ELSE
	(* server device not ready, reset local ready flag *)
	bReady := FALSE;
	nErrorId := BACnet_ERR_OPERATIONAL;
END_IF
(* set error flag *)
bError := (nErrorId <> BACnet_ERR_NO_ERROR);
END_FUNCTION_BLOCK

(* POU FB_BACnet_PulseConverter_RAW, ST *)
FUNCTION_BLOCK FB_BACnet_PulseConverter_RAW
VAR_INPUT
	nRawIn			AT%Q*: UINT; (* ~(BACnet_RawIoPulseConverterUnsignedValue : : ) *)
	bNoSensor		: BOOL;
	bOverRange		: BOOL;
	bUnderRange		: BOOL;
	bOpenLoop		: BOOL;
	bShortedLoop	: BOOL;
	bCommFailure	: BOOL;
	bConfigError	: BOOL;
	bOtherFault		: BOOL;
END_VAR
VAR_IN_OUT
	Device			: FB_BACnet_Device;
END_VAR
VAR_OUTPUT
	bReady			: BOOL;
	fPresentValue	: REAL;
	nCount			: UDINT;
	bOverridden		: BOOL;
	bOutOfService	: BOOL;
	bFault			: BOOL;
	bInAlarm		: BOOL;
	bError			: BOOL;
	nErrorId		: UINT;
END_VAR
VAR
	_PresentValueIn AT%I*: REAL; 	(* ~(BACnet_PresentValue 		:		: )
								   		(BACnet_ObjectType 			: PC	: )
										(BACnet_InputReference		: 		: nolink, disable) *)
	_Count AT%I*: UDINT;			(* ~(BACnet_Count		 		:		: ) *)
	_ObjectId AT%I*: DWORD;			(* ~(BACnet_ObjectIdentifier	:		: LINK) *)
	_StatusFlags AT%I*: WORD; 		(* ~(BACnet_StatusFlags 		:		: )	*)
	_ReliabilityIn AT%I*: WORD;		(* ~(BACnet_Reliability 		:		: )	*)
	_ReliabilityOut AT%Q*: WORD := BACnetReliability_no_fault_detected;(* ~(BACnet_Reliability 	:		: )	*)
	_StatusFlagsBits : ST_BACnet_StatusFlags;
	_nUpdateCount : UDINT := 0;
END_VAR
(* update server device *)
IF (Device._nUpdateCount = _nUpdateCount) THEN
	Device();
END_IF
(* remind current number of update counter *)
_nUpdateCount := Device._nUpdateCount;

(* handle raw error *)
IF (_ReliabilityIn <> BACnetReliability_configuration_error) THEN
	IF bNoSensor THEN
		_ReliabilityOut := BACnetReliability_no_sensor;
	ELSIF bOverRange THEN
		_ReliabilityOut := BACnetReliability_over_range;
	ELSIF bUnderRange THEN
		_ReliabilityOut := BACnetReliability_under_range;
	ELSIF bOpenLoop THEN
		_ReliabilityOut := BACnetReliability_open_loop;
	ELSIF bShortedLoop THEN
		_ReliabilityOut := BACnetReliability_shorted_loop;
	ELSIF bCommFailure THEN
		_ReliabilityOut := BACnetReliability_communication_failure;
	ELSIF bOtherFault THEN
		_ReliabilityOut := BACnetReliability_unreliable_other;
	ELSE
		_ReliabilityOut := BACnetReliability_no_fault_detected;
	END_IF
ELSE
	_ReliabilityOut := BACnetReliability_no_fault_detected;
END_IF

IF Device.bFirstCycle THEN
	(* first call of the server device since reboot/reset *)
	bReady := FALSE;

ELSIF (_StatusFlags < 4) THEN
	(* wrong mapping *)
	nErrorId := BACnet_ERR_WRONG_MAPPING;
	bReady := FALSE;

ELSIF Device.bOperational THEN
	(* ready state *)
	bReady := TRUE;
	nErrorId := BACnet_ERR_NO_ERROR;

	(* present value *)
	fPresentValue := _PresentValueIn;

	(* build bit states *)
	_StatusFlagsBits := F_BACnet_StatusFlags(_StatusFlags);

	(* copy states to output *)
	bOverridden		:= _StatusFlagsBits.overridden;
	bOutOfService	:= _StatusFlagsBits.out_of_service;
	bFault			:= _StatusFlagsBits.fault;
	bInAlarm		:= _StatusFlagsBits.in_alarm;

	(* additional information *)
	nCount			:= _Count;

ELSE
	(* server device not ready, reset local ready flag *)
	bReady := FALSE;
	nErrorId := BACnet_ERR_OPERATIONAL;
END_IF
(* set error flag *)
bError := (nErrorId <> BACnet_ERR_NO_ERROR);
END_FUNCTION_BLOCK

(* POU FB_BACnet_PWM, ST *)
FUNCTION_BLOCK FB_BACnet_PWM
VAR_INPUT
	bEnable			: BOOL;
	fPercent		: REAL; (* 0...100% *)
	tPeriod			: TIME; (* PWM period time *)
END_VAR
VAR_OUTPUT
	bEnablePV		: BOOL;
	bPresentValue	: BOOL;
END_VAR
VAR
	_fOut			: REAL;
	_tOn			: TIME;
	_tonPeriod		: TON;
	_tofOn			: TOF;
END_VAR
(* check limits *)
_fOut := LIMIT(0.0, fPercent, 100.0);

(* convert from percent value to time value in relation to period time (100% = tPara_Period, 0% = 0s) *)
_tOn := REAL_TO_TIME((_fOut / 100.0) * TIME_TO_REAL(tPeriod));

(* call period timer *)
_tonPeriod(
	IN	:= TRUE,
	PT	:= tPeriod,
	Q	=> ,
	ET	=> );

(* call on timer *)
_tofOn(
	IN	:= _tonPeriod.Q AND (_tOn > T#0ms),
	PT	:= _tOn,
	Q	=> ,
	ET	=> );

IF _tonPeriod.Q THEN
	_tonPeriod(IN:= FALSE);
	_tonPeriod(IN:= TRUE);
END_IF

(* set output *)
bPresentValue := (_tofOn.Q OR _tofOn.IN) AND bEnable;
bEnablePV := bEnable;
END_FUNCTION_BLOCK

(* POU FB_BACnet_RecipientListProperty, ST *)
FUNCTION_BLOCK FB_BACnet_RecipientListProperty
VAR_INPUT
	tObjectID			: T_BACnet_ObjectIdentifier := 16#FFFFFFFF;
	bAutoGet			: BOOL:=TRUE; (* TRUE = get data from property when ADS connection OR object ID changed *)
	bGet				: BOOL; (* FALSE --> TRUE = get data from property *)
	bSet				: BOOL; (* FALSE --> TRUE = set data into property *)
END_VAR
VAR_IN_OUT
	stAdsConn			: ST_BACnet_AdsConnection;
	stRecipients		: ST_BACnet_RecipientListDevice;
END_VAR
VAR_OUTPUT
	bDone				: BOOL;
	bBusy				: BOOL;
	bError				: BOOL;
	nErrorId			: UINT;
END_VAR
VAR
	_fbReadProp		: FB_BACnet_ReadProp;
	_fbWriteProp	: FB_BACnet_WriteProp;
	_i				: INT;
	_rtrigGet		: R_TRIG;
	_rtrigSet		: R_TRIG;

	_nAdsReloadOld	: USINT;
	_tObjectIDOld	: T_BACnet_ObjectIdentifier := 16#FFFFFFFF;

	_iEntryCheck	: UDINT;
	_iEntry			: INT;
	_iDataEntry		: INT;
	_iReadElems		: UDINT;

	_pEntryList		: POINTER TO T_BACnet_DestinationDeviceArray;

	_cbDestList		: UDINT;
	_cbDestListElem	: UDINT;
END_VAR
(*
	enum BACnetRecipient_Choice
	{
	      device,
	      address
	};
	
	typedef struct _BACnetObjectIdentifier
	{
	      union
	      {
	            struct 
	            {
	                  DWORD objInst : 22;
	                  DWORD objType : 10;
	            };
	            DWORD objId;
	      };
	}BACnetObjectIdentifier, *PBACnetObjectIdentifier;
	
	typedef struct _BACnetAddress
	{
	      BACnetAddressChoice choice;
	      BYTE layerAddress[7]; // MS/TP...LonTalk 
	      BYTE reserved;
	      USHORT      network_number;
	}BACnetAddress, *PBACnetAddress;
	
	enum BACnetAddressChoice
	{
	      Ethernet,
	      Arcnet,
	      MsTp,
	      LonTalk,
	      LonTalkNeuronId,
	      Address_3,
	      Address_4,
	      Address_5,
	      Broadcast
	};
	
	typedef struct _BACnetRecipient
	{ 
	      BACnetRecipient_Choice choiceField;
	      union
	      {
	            BACnetObjectIdentifier  device;
	            BACnetAddress           address;
	      };
	}BACnetRecipient,*PBACnetRecipient;
		
	typedef struct _BACnetDestination
	{ 
	      ULONG                              validDays;  //Bitfield of BACnetDaysOfWeek
	      BACnetTime                         fromTime;
	      BACnetTime                         toTime;
	      BACnetRecipient                    recipient;
	      ULONG                              processIdentifier;
	      DWORD                              transitionsBits;  // BACnetEventTransitionBits
	      BOOL                               issueConfirmedNotifications;
	}BACnetDestination,*PBACnetDestination;


*)

(* ADS read *)
_fbReadProp(
	BACnetDevicePort	:= stAdsConn.nAmsPort,
	bExecute			:= ,
	sNetId				:= stAdsConn.sAmsNetId,
	ObjectType			:= F_BACnet_GetObjType(tObjectID),
	PropertyID			:= BACnetPropertyIdentifier_RecipientList,
	DataType			:= BACnetDataType_RecipientArr,
	ObjectInstance		:= F_BACnet_GetObjInstance(tObjectID),
	ptrValue			:= ADR(stBACnet_AdsBuffer.arrData),
	nLenValue			:= SIZEOF(stBACnet_AdsBuffer.arrData),
	bDone				=> ,
	bBusy				=> ,
	bError				=> ,
	nErrID				=> ,
	nProcessedLen		=> );

(* ADS write *)
_fbWriteProp(
	BACnetDevicePort	:= stAdsConn.nAmsPort,
	bExecute			:= ,
	sNetId				:= stAdsConn.sAmsNetId,
	ObjectType			:= F_BACnet_GetObjType(tObjectID),
	PropertyID			:= BACnetPropertyIdentifier_RecipientList,
	Priority			:= BACnetPriority_None,
	DataType			:= BACnetDataType_RecipientArr,
	ObjectInstance		:= F_BACnet_GetObjInstance(tObjectID),
	ptrValue			:= ADR(stBACnet_AdsBuffer.arrData),
	nLenValue			:= _iDataEntry * _cbDestListElem,
	bDone				=> ,
	bBusy				=> ,
	bError				=> ,
	nErrID				=> );

(* trigger start event *)
_rtrigGet(CLK:= bGet, Q=> );
_rtrigSet(CLK:= bSet, Q=> );

(* state machine *)
CASE _i OF

	0: (* Idle *)
		IF 		_rtrigGet.Q
			OR	_rtrigSet.Q
			OR	(		(		(_nAdsReloadOld <> stAdsConn.nReload)
							OR	(_tObjectIDOld <> tObjectID)
						)
					AND	bAutoGet
				)
		THEN
			IF (NOT stAdsConn.bValid) THEN
				(* ADS connection not valid *)
				nErrorId := BACnet_ERR_INVALID_ADS_CONN;
			ELSE
				(* decide get or set *)
				IF _rtrigGet.Q THEN
					_i := 1;
				ELSIF _rtrigSet.Q THEN
					_i := 11;
				ELSIF bAutoGet THEN
					_i := 1;
				END_IF
				nErrorId := BACnet_ERR_NO_ERROR;
				(* reset index *)
				_iEntry	:= 0;
				(* initialize pointer *)
				_pEntryList := ADR(stBACnet_AdsBuffer.arrData);
				(* remind parameter *)
				_tObjectIDOld := tObjectID;
				_nAdsReloadOld := stAdsConn.nReload;
			END_IF
			(* reset done flag *)
			bDone := FALSE;
		END_IF
		IF (NOT bGet) AND (NOT bSet) AND (NOT bAutoGet) THEN
			nErrorId := BACnet_ERR_NO_ERROR;
			bDone := FALSE;
		END_IF

	(* READ *)
	1: (* read object property data via ADS *)
		IF TestAndSet(stBACnet_AdsBuffer.bTestSet) THEN
			IF _fbReadProp.bExecute THEN
				IF _fbReadProp.bError THEN
					_i := 100;
					nErrorId := BACnet_ERR_ADS_Read;
					_fbReadProp.bExecute := FALSE;
				ELSIF (NOT _fbReadProp.bBusy) THEN
					_i := 2;
					_fbReadProp.bExecute := FALSE;
					(* clear output data *)
					MEMSET(ADR(stRecipients), 0, SIZEOF(stRecipients));
					(* check array size *)
					_cbDestList 	:= SIZEOF(_pEntryList^);
					_cbDestListElem	:= SIZEOF(_pEntryList^[0]);
					_iEntryCheck := MIN(_fbReadProp.nProcessedLen, _cbDestList) MOD _cbDestListElem;
					IF (_iEntryCheck <> 0) OR (_cbDestListElem = 0) THEN
						_i := 100;
						nErrorId := BACnet_ERR_ADS_WrongEntrySize;
					ELSE
						(* scan property *)
						_iDataEntry := 0;
						_iReadElems := MIN(32767, MIN(_fbReadProp.nProcessedLen, _cbDestList) / _cbDestListElem);
						FOR _iEntry := 0 TO UDINT_TO_INT(_iReadElems) - 1 DO
							IF		(_pEntryList^[_iEntry].stRecipient.eRecipientChoice = BACnetRecipientChoice_device)
								AND	(F_BACnet_GetObjType(_pEntryList^[_iEntry].stRecipient.tDeviceId) = BACnetObjectType_Device)
							THEN
								stRecipients.arrDestList[_iDataEntry].stFromTime	:= _pEntryList^[_iEntry].stFromTime;
								stRecipients.arrDestList[_iDataEntry].stToTime	:= _pEntryList^[_iEntry].stToTime;
								stRecipients.arrDestList[_iDataEntry].tDeviceId	:= _pEntryList^[_iEntry].stRecipient.tDeviceId;
								stRecipients.arrDestList[_iDataEntry].nProcessId	:= _pEntryList^[_iEntry].nProcessId;
								stRecipients.arrDestList[_iDataEntry].bMonday		:= _F_BACnet_IsBitFieldBitSet(_pEntryList^[_iEntry].nValidDaysFlags, BACnetDaysOfWeekBits_Monday);
								stRecipients.arrDestList[_iDataEntry].bTuesday	:= _F_BACnet_IsBitFieldBitSet(_pEntryList^[_iEntry].nValidDaysFlags, BACnetDaysOfWeekBits_Tuesday);
								stRecipients.arrDestList[_iDataEntry].bWednesday	:= _F_BACnet_IsBitFieldBitSet(_pEntryList^[_iEntry].nValidDaysFlags, BACnetDaysOfWeekBits_Wednesday);
								stRecipients.arrDestList[_iDataEntry].bThursday	:= _F_BACnet_IsBitFieldBitSet(_pEntryList^[_iEntry].nValidDaysFlags, BACnetDaysOfWeekBits_Thursday);
								stRecipients.arrDestList[_iDataEntry].bFriday		:= _F_BACnet_IsBitFieldBitSet(_pEntryList^[_iEntry].nValidDaysFlags, BACnetDaysOfWeekBits_Friday);
								stRecipients.arrDestList[_iDataEntry].bSaturday	:= _F_BACnet_IsBitFieldBitSet(_pEntryList^[_iEntry].nValidDaysFlags, BACnetDaysOfWeekBits_Saturday);
								stRecipients.arrDestList[_iDataEntry].bSunday		:= _F_BACnet_IsBitFieldBitSet(_pEntryList^[_iEntry].nValidDaysFlags, BACnetDaysOfWeekBits_Sunday);
								stRecipients.arrDestList[_iDataEntry].bToNormal	:= _F_BACnet_IsBitFieldBitSet(_pEntryList^[_iEntry].nEventTransBits, BACnetEventTransitionBit_to_normal);
								stRecipients.arrDestList[_iDataEntry].bToOffNormal:= _F_BACnet_IsBitFieldBitSet(_pEntryList^[_iEntry].nEventTransBits, BACnetEventTransitionBit_to_offnormal);
								stRecipients.arrDestList[_iDataEntry].bToFault	:= _F_BACnet_IsBitFieldBitSet(_pEntryList^[_iEntry].nEventTransBits, BACnetEventTransitionBit_to_fault);
								stRecipients.arrDestList[_iDataEntry].bIssueConfirmedNotification	:= _pEntryList^[_iEntry].bIssueConfNot;
								_iDataEntry := _iDataEntry + 1;
							END_IF
						END_FOR
						(* calculate entry count *)
						stRecipients.nEntries := _iDataEntry;
						_i := 100;
					END_IF
				END_IF

			ELSIF (stBACnet_AdsBuffer.iLocked = 0) THEN
				_fbReadProp.bExecute := TRUE;
				(* lock global ADS buffer *)
				stBACnet_AdsBuffer.iLocked := SIZEOF(stBACnet_AdsBuffer.arrData);
			END_IF

			(* release temporary task lock *)
			stBACnet_AdsBuffer.bTestSet := FALSE;
		END_IF


	(* WRITE *)
	11: (* lock global ADS buffer *)
		IF TestAndSet(stBACnet_AdsBuffer.bTestSet) THEN
			IF stBACnet_AdsBuffer.iLocked = 0 THEN
				stBACnet_AdsBuffer.iLocked := SIZEOF(stBACnet_AdsBuffer.arrData);

				(* check array size *)
				_cbDestList 	:= SIZEOF(_pEntryList^);
				_cbDestListElem	:= SIZEOF(_pEntryList^[0]);

				(* scan property *)
				_iDataEntry := 0;
				FOR _iEntry := 0 TO MIN(stRecipients.nEntries - 1, BACnet_MaxDestinationArray) DO
					IF (F_BACnet_GetObjType(stRecipients.arrDestList[_iEntry].tDeviceId) = BACnetObjectType_Device) THEN
						(* clear buffer *)
						MEMSET(ADR(_pEntryList^[_iDataEntry]), 0, _cbDestListElem);
						(* copy time and recipient information *)
						_pEntryList^[_iDataEntry].stFromTime			:= stRecipients.arrDestList[_iEntry].stFromTime;
						_pEntryList^[_iDataEntry].stToTime				:= stRecipients.arrDestList[_iEntry].stToTime;
						_pEntryList^[_iDataEntry].stRecipient.tDeviceId	:= stRecipients.arrDestList[_iEntry].tDeviceId;
						_pEntryList^[_iDataEntry].nProcessId			:= stRecipients.arrDestList[_iEntry].nProcessId;
						(* set valid days flags *)
						_pEntryList^[_iDataEntry].nValidDaysFlags := DWORD#16#00000001;
						_F_BACnet_ChangeBitFieldBit(ADR(_pEntryList^[_iDataEntry].nValidDaysFlags), BACnetDaysOfWeekBits_Monday, stRecipients.arrDestList[_iEntry].bMonday);
						_F_BACnet_ChangeBitFieldBit(ADR(_pEntryList^[_iDataEntry].nValidDaysFlags), BACnetDaysOfWeekBits_Tuesday, stRecipients.arrDestList[_iEntry].bTuesday);
						_F_BACnet_ChangeBitFieldBit(ADR(_pEntryList^[_iDataEntry].nValidDaysFlags), BACnetDaysOfWeekBits_Wednesday, stRecipients.arrDestList[_iEntry].bWednesday);
						_F_BACnet_ChangeBitFieldBit(ADR(_pEntryList^[_iDataEntry].nValidDaysFlags), BACnetDaysOfWeekBits_Thursday, stRecipients.arrDestList[_iEntry].bThursday);
						_F_BACnet_ChangeBitFieldBit(ADR(_pEntryList^[_iDataEntry].nValidDaysFlags), BACnetDaysOfWeekBits_Friday, stRecipients.arrDestList[_iEntry].bFriday);
						_F_BACnet_ChangeBitFieldBit(ADR(_pEntryList^[_iDataEntry].nValidDaysFlags), BACnetDaysOfWeekBits_Saturday, stRecipients.arrDestList[_iEntry].bSaturday);
						_F_BACnet_ChangeBitFieldBit(ADR(_pEntryList^[_iDataEntry].nValidDaysFlags), BACnetDaysOfWeekBits_Sunday, stRecipients.arrDestList[_iEntry].bSunday);
						(* set event transition flags *)
						_pEntryList^[_iDataEntry].nEventTransBits := DWORD#16#00000005;
						_F_BACnet_ChangeBitFieldBit(ADR(_pEntryList^[_iDataEntry].nEventTransBits), BACnetEventTransitionBit_to_normal, stRecipients.arrDestList[_iEntry].bToNormal);
						_F_BACnet_ChangeBitFieldBit(ADR(_pEntryList^[_iDataEntry].nEventTransBits), BACnetEventTransitionBit_to_offnormal, stRecipients.arrDestList[_iEntry].bToOffNormal);
						_F_BACnet_ChangeBitFieldBit(ADR(_pEntryList^[_iDataEntry].nEventTransBits), BACnetEventTransitionBit_to_fault, stRecipients.arrDestList[_iEntry].bToFault);
						(* set confirmed notification flag *)
						_pEntryList^[_iDataEntry].bIssueConfNot := stRecipients.arrDestList[_iEntry].bIssueConfirmedNotification;
						(* set fix choice recipient choice *)
						_pEntryList^[_iDataEntry].stRecipient.eRecipientChoice := BACnetRecipientChoice_device;
						_iDataEntry := _iDataEntry + 1;
					ELSE
						(* Wrong recipient type (device expected) *)
						nErrorId := BACnet_ERR_ADS_RecipientData;
						_i := 100;
						EXIT;
					END_IF
				END_FOR
				(* send data *)
				_i := 12;
			END_IF
			(* release temporary task lock *)
			stBACnet_AdsBuffer.bTestSet := FALSE;
		END_IF

	12:
		IF _fbWriteProp.bExecute AND (NOT _fbWriteProp.bBusy) THEN
			(* check result *)
			_fbWriteProp.bExecute := FALSE;
			IF _fbWriteProp.bError THEN
				nErrorId := BACnet_ERR_ADS_Write;
			END_IF
			_i := 100;
		ELSE
			(* start ADS write *)
			_fbWriteProp.bExecute := TRUE;
		END_IF

	100: (* Done *)
		bDone := (nErrorId = BACnet_ERR_NO_ERROR);
		(* release ADS buffer *)
		stBACnet_AdsBuffer.iLocked := 0;
		_i := 0;

END_CASE

(* set error flag *)
bError 	:= nErrorId > BACnet_ERR_NO_ERROR;
bBusy 	:= _i > 0;
END_FUNCTION_BLOCK

(* POU FB_BACnet_RemoteAccumulator, ST *)
FUNCTION_BLOCK FB_BACnet_RemoteAccumulator
VAR_IN_OUT
	RemoteDevice		: FB_BACnet_RemoteDevice;
END_VAR
VAR_OUTPUT
	bReady				: BOOL;
	nPresentValue		: UDINT;
	bOverridden			: BOOL;
	bOutOfService		: BOOL;
	bFault				: BOOL;
	bInAlarm			: BOOL;
	bError				: BOOL;
	nErrorId			: UINT;
END_VAR
VAR
	_PresentValue AT%I*:UDINT;		(* ~(BACnet_PresentValue				:		: )
										(BACnet_ObjectType					: ACC	: )
										(BACnet_RemoteCycletimeRead			: 1000	: )
										(BACnet_RemoteFlagsRead				: 1		: )
										(BACnet_RemoteResubscriptionInterval: 240	: )
                                		(BACnet_RemoteCycleTimeWrite   		: 1000	: )
                                		(BACnet_RemoteFlagsWrite       		: 1		: )	*)
	_StatusFlags AT%I*:WORD;		(* ~(BACnet_StatusFlags					:		: )	*)
	_StatusFlagsBits : ST_BACnet_StatusFlags;

	_nUpdateCount : UDINT := 0;
END_VAR
(* update client device *)
IF RemoteDevice._nUpdateCount = _nUpdateCount THEN
	RemoteDevice();
END_IF
(* remind current number of update counter *)
_nUpdateCount := RemoteDevice._nUpdateCount;

IF NOT RemoteDevice.bOperational THEN
	nErrorId := BACnet_ERR_OPERATIONAL;
	bReady := FALSE;

ELSIF _StatusFlags >= 4 THEN
	(* clear error flag *)
	nErrorId := BACnet_ERR_NO_ERROR;
	bReady := TRUE;
	(* copy present value *)
	nPresentValue := _PresentValue;

	(* build bit states *)
	_StatusFlagsBits := F_BACnet_StatusFlags(_StatusFlags);

	(* copy states to output *)
	bOverridden := _StatusFlagsBits.overridden;
	bOutOfService := _StatusFlagsBits.out_of_service;
	bFault := _StatusFlagsBits.fault;
	bInAlarm := _StatusFlagsBits.in_alarm;
ELSE
	bReady := FALSE;
	(* and set error ID *)
	nErrorId := BACnet_ERR_WRONG_MAPPING;
END_IF

(* set error flag *)
bError := (nErrorId <> BACnet_ERR_NO_ERROR);
END_FUNCTION_BLOCK

(* POU FB_BACnet_RemoteDevice, ST *)
FUNCTION_BLOCK FB_BACnet_RemoteDevice
VAR_INPUT
	bReset				: BOOL;
	bAutoReset			: BOOL;
	bDisableWOC			: BOOL;
	bReSubscribeCOV		: BOOL;
	bAutoReSubscribe	: BOOL;
	bTriggerWOC			: BOOL; (* Revision 9 feature: FALSE --> TRUE writes all output process data to remote device *)
	nAmsPort			: UINT := 0; (* Optional setting: Ads port of BACnet client, default = not set *)
END_VAR
VAR_OUTPUT
	stAdsConn			: ST_BACnet_AdsConnection;
	eSystemStatus		: E_BACNETDEVICESTATUS;
	bEthLinkOk			: BOOL;
	bGatewayOk			: BOOL;
	sAmsNetId			: T_AmsNetId;
	bEnabledWOC			: BOOL;
	bWOCTriggered		: BOOL;
	bOperational		: BOOL;
	bConnecting			: BOOL;
	bFirstCycle			: BOOL;
	bError				: BOOL;
	nErrorId			: UINT;
	bClientTimeout		: BOOL;
	bServiceFailed		: BOOL;
	nTimeoutCnt			: UDINT;
	nServiceFailCnt		: UDINT;
END_VAR
VAR
	_ObjectId AT%I*:DWORD;			(* ~(BACnet_ObjectIdentifier			:		: LINK ) *)
	_SystemStatus AT%I*	: E_BACNETDEVICESTATUS;	(* ~
										(BACnet_SystemStatus 				: 		: )
										(BACnet_ObjectType					: DEV	: )
										(BACnet_RemoteCycletimeRead 		: 5000	: ) polling each 5 seconds
										(BACnet_RemoteFlagsRead        		: 2     : ) 2 = polling, so the object detects if the client is unreachable!
										(BACnet_RemoteResubscriptionInterval: 240 	: )
										(BACnet_RemoteCycleTimeWrite   		: 1000	: )
										(BACnet_RemoteFlagsWrite       		: 1		: ) *)
	_ClientStatus AT%I*:WORD;		(* ~(BACnet_ClientStatus				:		: )	*)
	_ClientControl AT%Q*:WORD;		(* ~(BACnet_ClientControl				:		: ) *)
	_rtrigReset			: R_TRIG;
	_rtrigOperational	: R_TRIG;
	_rtrigResubscribe	: R_TRIG;
	_rtrigTimeoutCnt	: R_TRIG;
	_rtrigServiceFailCnt: R_TRIG;
	_bReqResubscribe	: BOOL;
	_bComplete			: BOOL;
	_tofTimeoutLeft		: TOF;
	_tofServiceErrLeft	: TOF;
	_ftrigTimeoutLeft	: F_TRIG;

	_bHasStarted		: BOOL := TRUE;
	_nUpdateCount		: UDINT := 0;
	_nUpdateCountAdp 	: UDINT := 0;
	_BACnetAdapter		: POINTER TO FB_BACnet_Adapter;
	_AdsConn			: _FB_BACnet_AdsConn;
	_bLegacyMode		: BOOL;
	_tonAdsReset		: TON;

	_rtrigWOC			: R_TRIG;
	_bTriggerWOC		: BOOL;
	_tonWOCTrigger		: TON;
END_VAR
(* check pointer to bacnet adapter instance *)
IF pBACnet_Adapter > 0 THEN
	_BACnetAdapter := pBACnet_Adapter;
ELSE
	_BACnetAdapter := ADR(fbBACnet_Adapter);
END_IF

(* update server device *)
IF _BACnetAdapter^._nUpdateCount = _nUpdateCountAdp THEN
	_BACnetAdapter^();
END_IF
(* remind current number of update counter *)
_nUpdateCountAdp := _BACnetAdapter^._nUpdateCount;

(* check for client errors *)
_rtrigTimeoutCnt(CLK:= _ClientStatus.0, Q=> );
IF _rtrigTimeoutCnt.Q AND _bComplete THEN
	nErrorId := BACnet_ERR_CLIENT_TIMEOUT;
ELSIF (NOT _ClientStatus.0) THEN
	(* reset acknowledge flag *)
	_ClientControl.0 := FALSE;
END_IF
_rtrigServiceFailCnt(CLK:= _ClientStatus.1, Q=> );
IF _rtrigServiceFailCnt.Q AND _bComplete THEN
	nErrorId := BACnet_ERR_CLIENT_SERVICE;
ELSIF (NOT _ClientStatus.1) THEN
	(* reset acknowledge flag *)
	_ClientControl.1 := FALSE;
END_IF

(* convert SystemStatus to enumeration *)
eSystemStatus := _SystemStatus;
(* reset trigger *)
_rtrigReset(CLK:= bReset, Q=> );
(* reset error ID and flag *)
IF (nErrorId < 20) OR _rtrigReset.Q OR bAutoReset THEN
	nErrorId := BACnet_ERR_NO_ERROR;
END_IF
IF _rtrigReset.Q OR (NOT _bComplete) OR bAutoReset THEN
	_ClientControl.0 := _ClientStatus.0;
	_ClientControl.1 := _ClientStatus.1;
END_IF

(* read NetId and convert to string *)
sAmsNetId := _BACnetAdapter^.sAmsNetId;
(* check if it plausible *)
IF sAmsNetId = '' THEN
	(* NetId not OK, return with error *)
	nErrorId := BACnet_ERR_NO_VALID_NET_ID;
ELSIF (NOT _BACnetAdapter^.bEthLinkOk) THEN
	(* ethernet link missing *)
	nErrorId := BACnet_ERR_NO_ETH_LINK;
ELSIF (NOT _BACnetAdapter^.bGatewayOk) THEN
	(* gateway missing *)
	nErrorId := BACnet_ERR_NO_GATEWAY;
END_IF

(* summerize timeout errors *)
_tofTimeoutLeft(
	IN:= (_rtrigTimeoutCnt.Q AND _bComplete),
	PT:= T#20s,
	Q=> bClientTimeout,
	ET=> );
IF _tofTimeoutLeft.IN THEN
	nTimeoutCnt := nTimeoutCnt + 1;
END_IF
_ftrigTimeoutLeft(CLK:= _tofTimeoutLeft.Q, Q=> );

(* summerize service errors *)
_tofServiceErrLeft(
	IN:= (_rtrigServiceFailCnt.Q AND _bComplete),
	PT:= T#20s,
	Q=> bServiceFailed,
	ET=> );
IF _tofServiceErrLeft.IN THEN
	nServiceFailCnt := nServiceFailCnt + 1;
END_IF

(* WOC trigger control *)
_rtrigWOC(CLK:= bTriggerWOC, Q=> );
IF (_ClientStatus.2 OR bDisableWOC) AND bTriggerWOC THEN
	nErrorId := BACnet_ERR_WOC_DISABLED;
	_bTriggerWOC := FALSE;
ELSIF _ClientStatus.4 OR _bTriggerWOC THEN
	IF _rtrigWOC.Q THEN
		nErrorId := BACnet_ERR_WOC_TRIGGER_ACTIVE;
	ELSIF (NOT bTriggerWOC) THEN
		_bTriggerWOC := FALSE;
	END_IF
ELSIF _rtrigWOC.Q THEN
	_bTriggerWOC := TRUE;
END_IF

(* controls *)
_ClientControl.2 := bDisableWOC;
_ClientControl.3 := _bReqResubscribe;
_ClientControl.4 := _bTriggerWOC;

(* states *)
bEthLinkOk := _BACnetAdapter^.bEthLinkOk;
bGatewayOk := _BACnetAdapter^.bGatewayOk;

bEnabledWOC := (NOT _ClientStatus.2);
bConnecting := (SHR((_ClientStatus AND 16#FF00), 8) < 4);
_bComplete :=		(NOT bConnecting)
				AND	(_SystemStatus = 0)
				AND	_BACnetAdapter^.bEthLinkOk;
bOperational :=		_bComplete
				AND ((NOT _ClientStatus.0) OR bAutoReset);
bWOCTriggered	:= bTriggerWOC AND _ClientStatus.4 AND (NOT (_ClientStatus.2 OR bDisableWOC));

(* Resubscribe COV *)
_rtrigOperational(CLK:= bOperational, Q=> );
_rtrigResubscribe(CLK:= bReSubscribeCOV, Q=> );
IF		(		(		(		_rtrigOperational.Q
							OR (_ftrigTimeoutLeft.Q AND bAutoReset)
						)
					AND	bAutoReSubscribe
				)
			OR	_rtrigResubscribe.Q
		)
	AND	(NOT _bReqResubscribe)
THEN
	(* operation mode reached or resubscription was externally triggered, start resubcription *)
	_bReqResubscribe	:= TRUE;
ELSIF (NOT bOperational) THEN
	(* not operational *)
	_bReqResubscribe	:= FALSE;
ELSE
	IF _bReqResubscribe AND _ClientStatus.3 THEN
		(* resubscription triggered *)
		_bReqResubscribe := FALSE;
	END_IF
END_IF

(* check WOC trigger state *)
_tonWOCTrigger(IN:= _bTriggerWOC, PT:= T#5s, Q=> , ET=> );
IF _tonWOCTrigger.Q THEN
	nErrorId := BACnet_ERR_WOC_TRIGGER_UNSUP;
	IF (NOT bTriggerWOC) THEN
		_bTriggerWOC := FALSE;
	END_IF
END_IF

IF (NOT _bLegacyMode) AND _bComplete AND (_ObjectId <> 0) THEN
	(* call ADS connection *)
	_AdsConn(
		bAutoReload		:= TRUE,
		bReload			:=	(bReset AND (NOT _AdsConn.bReady) AND (NOT bAutoReset))
						OR	_tonAdsReset.Q
						OR	_ftrigTimeoutLeft.Q,
		bIsClient		:= TRUE,
		bDevOperational	:= bOperational,
		sAmsNetId		:= sAmsNetId,
		tDevObjId		:= _ObjectId,
		bReady			=> ,
		bBusy			=> ,
		bDone			=> ,
		bError			=> ,
		nErrorId		=> ,
		stBACnetAds		=> stAdsConn);

	(* error when ADS connection failed *)
	IF _AdsConn.bError THEN
		IF (_AdsConn.nErrorId = BACnet_ERR_ADS_LegacyStack) THEN
			_bLegacyMode := TRUE;
		ELSIF (nErrorId = 0) THEN
			nErrorId := _AdsConn.nErrorId;
		END_IF
	END_IF

	(* auto reload when error is active *)
	_tonAdsReset(
		IN:=	(NOT _AdsConn.bReload)
			AND	_AdsConn.bError
			AND	bAutoReset
			AND bOperational,
		PT:= t#2s,
		Q=> ,
		ET=> );
END_IF
IF _bLegacyMode THEN
	stAdsConn.bClient	:= TRUE;
	stAdsConn.bServer	:= FALSE;
	stAdsConn.bValid	:= FALSE;
	stAdsConn.nAmsPort	:= nAmsPort;
	stAdsConn.sAmsNetId	:= sAmsNetId;
	stAdsConn.nDeviceId	:= F_BACnet_GetObjInstance(_ObjectId);
END_IF


bError := (nErrorId <> BACnet_ERR_NO_ERROR);

(* update counter *)
IF (_nUpdateCount = 0) AND _bHasStarted THEN
	bFirstCycle := TRUE;
	_bHasStarted := FALSE;
ELSE
	bFirstCycle := FALSE;
END_IF
_nUpdateCount := _nUpdateCount + 1;
END_FUNCTION_BLOCK

(* POU FB_BACnet_RemoteAccumulator_EX, ST *)
FUNCTION_BLOCK FB_BACnet_RemoteAccumulator_EX
VAR_IN_OUT
	RemoteDevice		: FB_BACnet_RemoteDevice;
END_VAR
VAR_OUTPUT
	bReady				: BOOL;
	nPresentValue		: UDINT;
	bOverridden			: BOOL;
	bOutOfService		: BOOL;
	bFault				: BOOL;
	bInAlarm			: BOOL;
	bOverRange			: BOOL;
	bUnderRange			: BOOL;
	bNoSensor			: BOOL;
	bOpenLoop			: BOOL;
	bCommFailure		: BOOL;
	bShortedLoop		: BOOL;
	bOtherFault			: BOOL;
	tObjectID			: T_BACnet_ObjectIdentifier := 16#FFFFFFFF;
	bError				: BOOL;
	nErrorId			: UINT;
END_VAR
VAR
	_PresentValue AT%I*:UDINT;			(* ~(BACnet_PresentValue				:		: )
											(BACnet_ObjectType					: ACC	: )
											(BACnet_RemoteCycletimeRead			: 1000	: )
											(BACnet_RemoteFlagsRead				: 1		: )
											(BACnet_RemoteResubscriptionInterval: 240	: )
                                			(BACnet_RemoteCycleTimeWrite   		: 1000	: )
                                			(BACnet_RemoteFlagsWrite       		: 1		: )	*)
	_ObjectId AT%I*: DWORD;				(* ~(BACnet_ObjectIdentifier			:		: LINK) *)
	_StatusFlags AT%I*:WORD;			(* ~(BACnet_StatusFlags					:		: )	*)
	_Reliability AT%I*:WORD;			(* ~(BACnet_Reliability					:		: )	*)
	_StatusFlagsBits : ST_BACnet_StatusFlags;

	_nUpdateCount : UDINT := 0;
END_VAR
(* update client device *)
IF RemoteDevice._nUpdateCount = _nUpdateCount THEN
	RemoteDevice();
END_IF
(* remind current number of update counter *)
_nUpdateCount := RemoteDevice._nUpdateCount;

IF NOT RemoteDevice.bOperational THEN
	nErrorId := BACnet_ERR_OPERATIONAL;
	bReady := FALSE;

ELSIF (F_BACnet_GetObjType(_ObjectId) <> BACnetObjectType_Accumulator) THEN
	(* wrong mapping / invalid object ID *)
	IF _ObjectId = 0 THEN
		nErrorId := BACnet_ERR_WRONG_MAPPING;
	ELSE
		nErrorId := BACnet_ERR_INVALID_OBJECTID;
	END_IF
	bReady := FALSE;
	tObjectID := 16#FFFFFFFF;

ELSIF _StatusFlags >= 4 THEN
	(* clear error flag *)
	nErrorId := BACnet_ERR_NO_ERROR;
	bReady := TRUE;
	(* copy present value *)
	nPresentValue := _PresentValue;

	(* build bit states *)
	_StatusFlagsBits := F_BACnet_StatusFlags(_StatusFlags);

	(* copy states to output *)
	bOverridden := _StatusFlagsBits.overridden;
	bOutOfService := _StatusFlagsBits.out_of_service;
	bFault := _StatusFlagsBits.fault;
	bInAlarm := _StatusFlagsBits.in_alarm;
	bOverRange := (_Reliability = BACnetReliability_over_range);
	bUnderRange := (_Reliability = BACnetReliability_under_range);
	bNoSensor := (_Reliability = BACnetReliability_no_sensor);
	bOpenLoop := (_Reliability = BACnetReliability_open_loop);
	bCommFailure := (_Reliability = BACnetReliability_communication_failure);
	bShortedLoop := (_Reliability = BACnetReliability_shorted_loop);
	bOtherFault := (_Reliability = BACnetReliability_unreliable_other);
	tObjectID := _ObjectId;

ELSE
	bReady := FALSE;
	(* and set error ID *)
	nErrorId := BACnet_ERR_WRONG_MAPPING;
END_IF

(* set error flag *)
bError := (nErrorId <> BACnet_ERR_NO_ERROR);
END_FUNCTION_BLOCK

(* POU FB_BACnet_RemoteAccumulator_POLL, ST *)
FUNCTION_BLOCK FB_BACnet_RemoteAccumulator_POLL
VAR_IN_OUT
	RemoteDevice		: FB_BACnet_RemoteDevice;
END_VAR
VAR_OUTPUT
	bReady				: BOOL;
	nPresentValue		: UDINT;
	bOverridden			: BOOL;
	bOutOfService		: BOOL;
	bFault				: BOOL;
	bInAlarm			: BOOL;
	bError				: BOOL;
	nErrorId			: UINT;
END_VAR
VAR
	_PresentValue AT%I*:UDINT;		(* ~(BACnet_PresentValue				:		: )
										(BACnet_ObjectType					: ACC	: )
										(BACnet_RemoteCycletimeRead			: 5000	: )
										(BACnet_RemoteFlagsRead				: 2		: )
                                		(BACnet_RemoteCycleTimeWrite   		: 1000	: )
                                		(BACnet_RemoteFlagsWrite       		: 1		: )	*)
	_StatusFlags AT%I*:WORD;		(* ~(BACnet_StatusFlags					:		: )	*)
	_StatusFlagsBits : ST_BACnet_StatusFlags;

	_nUpdateCount : UDINT := 0;
END_VAR
(* update client device *)
IF RemoteDevice._nUpdateCount = _nUpdateCount THEN
	RemoteDevice();
END_IF
(* remind current number of update counter *)
_nUpdateCount := RemoteDevice._nUpdateCount;

IF NOT RemoteDevice.bOperational THEN
	nErrorId := BACnet_ERR_OPERATIONAL;
	bReady := FALSE;

ELSIF _StatusFlags >= 4 THEN
	(* clear error flag *)
	nErrorId := BACnet_ERR_NO_ERROR;
	bReady := TRUE;
	(* copy present value *)
	nPresentValue := _PresentValue;

	(* build bit states *)
	_StatusFlagsBits := F_BACnet_StatusFlags(_StatusFlags);

	(* copy states to output *)
	bOverridden := _StatusFlagsBits.overridden;
	bOutOfService := _StatusFlagsBits.out_of_service;
	bFault := _StatusFlagsBits.fault;
	bInAlarm := _StatusFlagsBits.in_alarm;
ELSE
	bReady := FALSE;
	(* and set error ID *)
	nErrorId := BACnet_ERR_WRONG_MAPPING;
END_IF

(* set error flag *)
bError := (nErrorId <> BACnet_ERR_NO_ERROR);
END_FUNCTION_BLOCK

(* POU FB_BACnet_RemoteAnalogInput, ST *)
FUNCTION_BLOCK FB_BACnet_RemoteAnalogInput
VAR_IN_OUT
	RemoteDevice			: FB_BACnet_RemoteDevice;
END_VAR
VAR_OUTPUT
	bReady				: BOOL;
	fPresentValue		: REAL;
	bOverridden			: BOOL;
	bOutOfService		: BOOL;
	bFault				: BOOL;
	bInAlarm			: BOOL;
	bError				: BOOL;
	nErrorId			: UINT;
END_VAR
VAR
	_PresentValue AT%I*: REAL; 			(* ~(BACnet_PresentValue 				:		: )
								   			(BACnet_ObjectType 					: AI	: )
											(BACnet_RemoteCycletimeRead 		: 1000	: )
											(BACnet_RemoteFlagsRead        		: 1		: )
											(BACnet_RemoteResubscriptionInterval: 240	: )
	                                		(BACnet_RemoteCycleTimeWrite   		: 1000	: )
	                                		(BACnet_RemoteFlagsWrite       		: 1		: )	*)
	_StatusFlags AT%I*: WORD; 			(* ~(BACnet_StatusFlags 				:		: )	*)
	_StatusFlagsBits : ST_BACnet_StatusFlags;

	_nUpdateCount : UDINT := 0;
END_VAR
(* update client device *)
IF RemoteDevice._nUpdateCount = _nUpdateCount THEN
	RemoteDevice();
END_IF
(* remind current number of update counter *)
_nUpdateCount := RemoteDevice._nUpdateCount;

IF NOT RemoteDevice.bOperational THEN
	nErrorId := BACnet_ERR_OPERATIONAL;
	bReady := FALSE;

ELSIF _StatusFlags >= 4 THEN
	(* clear error flag *)
	nErrorId := BACnet_ERR_NO_ERROR;
	(* ready state *)
	bReady := TRUE;

	(* present value *)
	fPresentValue := _PresentValue;

	(* build bit states *)
	_StatusFlagsBits := F_BACnet_StatusFlags(_StatusFlags);

	(* copy states to output *)
	bOverridden := _StatusFlagsBits.overridden;
	bOutOfService := _StatusFlagsBits.out_of_service;
	bFault := _StatusFlagsBits.fault;
	bInAlarm := _StatusFlagsBits.in_alarm;
ELSE
	(* server device not ready, reset local ready also *)
	bReady := FALSE;
	(* and set error ID *)
	nErrorId := BACnet_ERR_WRONG_MAPPING;
END_IF

(* set error flag *)
bError := (nErrorId <> BACnet_ERR_NO_ERROR);
END_FUNCTION_BLOCK

(* POU FB_BACnet_RemoteAnalogInput_EX, ST *)
FUNCTION_BLOCK FB_BACnet_RemoteAnalogInput_EX
VAR_IN_OUT
	RemoteDevice			: FB_BACnet_RemoteDevice;
END_VAR
VAR_OUTPUT
	bReady				: BOOL;
	fPresentValue		: REAL;
	bOverridden			: BOOL;
	bOutOfService		: BOOL;
	bFault				: BOOL;
	bInAlarm			: BOOL;
	bOverRange			: BOOL;
	bUnderRange			: BOOL;
	bNoSensor			: BOOL;
	bOpenLoop			: BOOL;
	bShortedLoop		: BOOL;
	bOtherFault			: BOOL;
	eEventState			: E_BACNETEVENTSTATE;
	tObjectID			: T_BACnet_ObjectIdentifier := 16#FFFFFFFF;
	bError				: BOOL;
	nErrorId			: UINT;
END_VAR
VAR
	_PresentValue AT%I*: REAL; 			(* ~(BACnet_PresentValue 				:		: )
								   			(BACnet_ObjectType 					: AI	: )
											(BACnet_RemoteCycletimeRead 		: 1000	: )
											(BACnet_RemoteFlagsRead        		: 1		: )
											(BACnet_RemoteResubscriptionInterval: 240	: )
	                                		(BACnet_RemoteCycleTimeWrite   		: 1000	: )
	                                		(BACnet_RemoteFlagsWrite       		: 1		: )	*)
	_ObjectId AT%I*: DWORD;				(* ~(BACnet_ObjectIdentifier			:		: LINK) *)
	_StatusFlags AT%I*: WORD; 			(* ~(BACnet_StatusFlags 				:		: )	*)
	_Reliability AT%I*: WORD; 			(* ~(BACnet_Reliability 				:		: )	*)
	_EventState AT%I*: WORD;			(* ~(BACnet_EventState					:		: )	*)
	_nUpdateCount : UDINT := 0;
	_StatusFlagsBits : ST_BACnet_StatusFlags;
END_VAR
(* update client device *)
IF RemoteDevice._nUpdateCount = _nUpdateCount THEN
	RemoteDevice();
END_IF
(* remind current number of update counter *)
_nUpdateCount := RemoteDevice._nUpdateCount;

IF NOT RemoteDevice.bOperational THEN
	nErrorId := BACnet_ERR_OPERATIONAL;
	bReady := FALSE;

ELSIF (F_BACnet_GetObjType(_ObjectId) <> BACnetObjectType_AnalogInput) THEN
	(* wrong mapping / invalid object ID *)
	IF _ObjectId = 0 THEN
		nErrorId := BACnet_ERR_WRONG_MAPPING;
	ELSE
		nErrorId := BACnet_ERR_INVALID_OBJECTID;
	END_IF
	bReady := FALSE;
	tObjectID := 16#FFFFFFFF;

ELSIF _StatusFlags >= 4 THEN
	(* clear error flag *)
	nErrorId := BACnet_ERR_NO_ERROR;
	(* ready state *)
	bReady := TRUE;

	(* present value *)
	fPresentValue := _PresentValue;

	(* build bit states *)
	_StatusFlagsBits := F_BACnet_StatusFlags(_StatusFlags);

	(* copy states to output *)
	bOverridden := _StatusFlagsBits.overridden;
	bOutOfService := _StatusFlagsBits.out_of_service;
	bFault := _StatusFlagsBits.fault;
	bInAlarm := _StatusFlagsBits.in_alarm;
	bOverRange := (_Reliability = BACnetReliability_over_range);
	bUnderRange := (_Reliability = BACnetReliability_under_range);
	bNoSensor := (_Reliability = BACnetReliability_no_sensor);
	bOpenLoop := (_Reliability = BACnetReliability_open_loop);
	bShortedLoop := (_Reliability = BACnetReliability_shorted_loop);
	bOtherFault := (_Reliability = BACnetReliability_unreliable_other);
	eEventState := _EventState;
	tObjectID := _ObjectId;
ELSE
	(* server device not ready, reset local ready also *)
	bReady := FALSE;
	(* and set error ID *)
	nErrorId := BACnet_ERR_WRONG_MAPPING;
END_IF

(* set error flag *)
bError := (nErrorId <> BACnet_ERR_NO_ERROR);
END_FUNCTION_BLOCK

(* POU FB_BACnet_RemoteAnalogInput_POLL, ST *)
FUNCTION_BLOCK FB_BACnet_RemoteAnalogInput_POLL
VAR_IN_OUT
	RemoteDevice			: FB_BACnet_RemoteDevice;
END_VAR
VAR_OUTPUT
	bReady				: BOOL;
	fPresentValue		: REAL;
	bOverridden			: BOOL;
	bOutOfService		: BOOL;
	bFault				: BOOL;
	bInAlarm			: BOOL;
	bError				: BOOL;
	nErrorId			: UINT;
END_VAR
VAR
	_PresentValue AT%I*: REAL; 			(* ~(BACnet_PresentValue 				:		: )
								   			(BACnet_ObjectType 					: AI	: )
											(BACnet_RemoteCycletimeRead 		: 5000	: )
											(BACnet_RemoteFlagsRead        		: 2		: )
	                                		(BACnet_RemoteCycleTimeWrite   		: 1000	: )
	                                		(BACnet_RemoteFlagsWrite       		: 1		: )	*)
	_StatusFlags AT%I*: WORD; 			(* ~(BACnet_StatusFlags 				:		: )	*)
	_StatusFlagsBits : ST_BACnet_StatusFlags;

	_nUpdateCount : UDINT := 0;
END_VAR
(* update client device *)
IF RemoteDevice._nUpdateCount = _nUpdateCount THEN
	RemoteDevice();
END_IF
(* remind current number of update counter *)
_nUpdateCount := RemoteDevice._nUpdateCount;

IF NOT RemoteDevice.bOperational THEN
	nErrorId := BACnet_ERR_OPERATIONAL;
	bReady := FALSE;

ELSIF _StatusFlags >= 4 THEN
	(* clear error flag *)
	nErrorId := BACnet_ERR_NO_ERROR;
	(* ready state *)
	bReady := TRUE;

	(* present value *)
	fPresentValue := _PresentValue;

	(* build bit states *)
	_StatusFlagsBits := F_BACnet_StatusFlags(_StatusFlags);

	(* copy states to output *)
	bOverridden := _StatusFlagsBits.overridden;
	bOutOfService := _StatusFlagsBits.out_of_service;
	bFault := _StatusFlagsBits.fault;
	bInAlarm := _StatusFlagsBits.in_alarm;
ELSE
	(* server device not ready, reset local ready also *)
	bReady := FALSE;
	(* and set error ID *)
	nErrorId := BACnet_ERR_WRONG_MAPPING;
END_IF

(* set error flag *)
bError := (nErrorId <> BACnet_ERR_NO_ERROR);
END_FUNCTION_BLOCK

(* POU FB_BACnet_RemoteAnalogOutput, ST *)
FUNCTION_BLOCK FB_BACnet_RemoteAnalogOutput
VAR_INPUT
	bEnablePV		: BOOL; (* enable present value with priority x in priority array, FALSE = priority x disable *)
	fPV		: REAL; (* decimal number for priority x, when input bEnablePV is TRUE *)
END_VAR
VAR_IN_OUT
	RemoteDevice	: FB_BACnet_RemoteDevice;
END_VAR
VAR_OUTPUT
	bReady				: BOOL;
	fPresentValue		: REAL;
	bOverridden			: BOOL;
	bOutOfService		: BOOL;
	bFault				: BOOL;
	bInAlarm			: BOOL;
	bError				: BOOL;
	nErrorId			: UINT;
END_VAR
VAR
	_PresentValue AT%I*: REAL; 			(* ~(BACnet_PresentValue 				:		: )
								   			(BACnet_ObjectType 					: AO	: )
											(BACnet_RemoteCycletimeRead 		: 1000	: )
											(BACnet_RemoteFlagsRead        		: 1		: )
											(BACnet_RemoteResubscriptionInterval: 240	: )
	                                		(BACnet_RemoteCycleTimeWrite   		: 1000	: )
	                                		(BACnet_RemoteFlagsWrite       		: 1		: )	*)
    _PresentValue_Priority12 AT%Q*: REAL;(* ~(BACnet_PresentValue_Priority12	:		: )	*)
	_StatusFlags AT%I*: WORD; 			(* ~(BACnet_StatusFlags 				:		: )	*)
	_StatusFlagsBits : ST_BACnet_StatusFlags;

	_nUpdateCount : UDINT := 0;
END_VAR
(* update client device *)
IF RemoteDevice._nUpdateCount = _nUpdateCount THEN
	RemoteDevice();
END_IF
(* remind current number of update counter *)
_nUpdateCount := RemoteDevice._nUpdateCount;

IF RemoteDevice.bFirstCycle THEN
	(* first call of the server device since reboot/reset *)
	bReady := FALSE;
	_PresentValue_Priority12 := F_BACnet_NAN();
ELSIF NOT RemoteDevice.bOperational THEN
	nErrorId := BACnet_ERR_OPERATIONAL;
	bReady := FALSE;

ELSIF _StatusFlags >= 4 THEN
	(* clear error flag *)
	nErrorId := BACnet_ERR_NO_ERROR;
	(* ready state *)
	bReady := TRUE;

	(* write into priority array *)
	IF bEnablePV THEN
		_PresentValue_Priority12	:= fPV;
	ELSE
		_PresentValue_Priority12	:= F_BACnet_NAN();
	END_IF

	(* present value *)
	fPresentValue := _PresentValue;

	(* build bit states *)
	_StatusFlagsBits := F_BACnet_StatusFlags(_StatusFlags);

	(* copy states to output *)
	bOverridden := _StatusFlagsBits.overridden;
	bOutOfService := _StatusFlagsBits.out_of_service;
	bFault := _StatusFlagsBits.fault;
	bInAlarm := _StatusFlagsBits.in_alarm;
ELSE
	(* server device not ready, reset local ready also *)
	bReady := FALSE;
	(* and set error ID *)
	nErrorId := BACnet_ERR_WRONG_MAPPING;
END_IF

(* set error flag *)
bError := (nErrorId <> BACnet_ERR_NO_ERROR);
END_FUNCTION_BLOCK

(* POU FB_BACnet_RemoteAnalogOutput_EX, ST *)
FUNCTION_BLOCK FB_BACnet_RemoteAnalogOutput_EX
VAR_INPUT
	bEnablePV		: BOOL; (* enable present value with priority x in priority array, FALSE = priority x disable *)
	fPV		: REAL; (* decimal number for priority x, when input bEnablePV is TRUE *)
END_VAR
VAR_IN_OUT
	RemoteDevice	: FB_BACnet_RemoteDevice;
END_VAR
VAR_OUTPUT
	bReady				: BOOL;
	fPresentValue		: REAL;
	bOverridden			: BOOL;
	bOutOfService		: BOOL;
	bFault				: BOOL;
	bInAlarm			: BOOL;
	bNoOutput			: BOOL;
	bOpenLoop			: BOOL;
	bShortedLoop		: BOOL;
	bOtherFault			: BOOL;
	eEventState			: E_BACNETEVENTSTATE;
	tObjectID			: T_BACnet_ObjectIdentifier := 16#FFFFFFFF;
	bError				: BOOL;
	nErrorId			: UINT;
END_VAR
VAR
	_PresentValue AT%I*: REAL; 			(* ~(BACnet_PresentValue 				:		: )
								   			(BACnet_ObjectType 					: AO	: )
											(BACnet_RemoteCycletimeRead 		: 1000	: )
											(BACnet_RemoteFlagsRead        		: 1		: )
											(BACnet_RemoteResubscriptionInterval: 240	: )
	                                		(BACnet_RemoteCycleTimeWrite   		: 1000	: )
	                                		(BACnet_RemoteFlagsWrite       		: 1		: )	*)
    _PresentValue_Priority12 AT%Q*: REAL;(* ~(BACnet_PresentValue_Priority12	:		: )	*)
	_ObjectId AT%I*: DWORD;				(* ~(BACnet_ObjectIdentifier			:		: LINK) *)
	_StatusFlags AT%I*: WORD; 			(* ~(BACnet_StatusFlags 				:		: )	*)
	_Reliability AT%I*: WORD; 			(* ~(BACnet_Reliability 				:		: )	*)
	_EventState AT%I*: WORD;			(* ~(BACnet_EventState					:		: )	*)
	_nUpdateCount : UDINT := 0;
	_StatusFlagsBits : ST_BACnet_StatusFlags;
END_VAR
(* update client device *)
IF RemoteDevice._nUpdateCount = _nUpdateCount THEN
	RemoteDevice();
END_IF
(* remind current number of update counter *)
_nUpdateCount := RemoteDevice._nUpdateCount;

IF RemoteDevice.bFirstCycle THEN
	(* first call of the server device since reboot/reset *)
	bReady := FALSE;
	_PresentValue_Priority12 := F_BACnet_NAN();

ELSIF NOT RemoteDevice.bOperational THEN
	nErrorId := BACnet_ERR_OPERATIONAL;
	bReady := FALSE;

ELSIF (F_BACnet_GetObjType(_ObjectId) <> BACnetObjectType_AnalogOutput) THEN
	(* wrong mapping / invalid object ID *)
	IF _ObjectId = 0 THEN
		nErrorId := BACnet_ERR_WRONG_MAPPING;
	ELSE
		nErrorId := BACnet_ERR_INVALID_OBJECTID;
	END_IF
	bReady := FALSE;
	tObjectID := 16#FFFFFFFF;

ELSIF _StatusFlags >= 4 THEN
	(* clear error flag *)
	nErrorId := BACnet_ERR_NO_ERROR;
	(* ready state *)
	bReady := TRUE;

	(* write into priority array *)
	IF bEnablePV THEN
		_PresentValue_Priority12	:= fPV;
	ELSE
		_PresentValue_Priority12	:= F_BACnet_NAN();
	END_IF

	(* present value *)
	fPresentValue := _PresentValue;

	(* build bit states *)
	_StatusFlagsBits := F_BACnet_StatusFlags(_StatusFlags);

	(* copy states to output *)
	bOverridden := _StatusFlagsBits.overridden;
	bOutOfService := _StatusFlagsBits.out_of_service;
	bFault := _StatusFlagsBits.fault;
	bInAlarm := _StatusFlagsBits.in_alarm;
	bNoOutput := (_Reliability = BACnetReliability_no_output);
	bOpenLoop := (_Reliability = BACnetReliability_open_loop);
	bShortedLoop := (_Reliability = BACnetReliability_shorted_loop);
	bOtherFault := (_Reliability = BACnetReliability_unreliable_other);
	eEventState := _EventState;
	tObjectID := _ObjectId;
ELSE
	(* server device not ready, reset local ready also *)
	bReady := FALSE;
	(* and set error ID *)
	nErrorId := BACnet_ERR_WRONG_MAPPING;
END_IF

(* set error flag *)
bError := (nErrorId <> BACnet_ERR_NO_ERROR);
END_FUNCTION_BLOCK

(* POU FB_BACnet_RemoteAnalogOutput_POLL, ST *)
FUNCTION_BLOCK FB_BACnet_RemoteAnalogOutput_POLL
VAR_INPUT
	bEnablePV		: BOOL; (* enable present value with priority x in priority array, FALSE = priority x disable *)
	fPV		: REAL; (* decimal number for priority x, when input bEnablePV is TRUE *)
END_VAR
VAR_IN_OUT
	RemoteDevice	: FB_BACnet_RemoteDevice;
END_VAR
VAR_OUTPUT
	bReady				: BOOL;
	fPresentValue		: REAL;
	bOverridden			: BOOL;
	bOutOfService		: BOOL;
	bFault				: BOOL;
	bInAlarm			: BOOL;
	bError				: BOOL;
	nErrorId			: UINT;
END_VAR
VAR
	_PresentValue AT%I*: REAL; 			(* ~(BACnet_PresentValue 				:		: )
								   			(BACnet_ObjectType 					: AO	: )
											(BACnet_RemoteCycletimeRead 		: 5000	: )
											(BACnet_RemoteFlagsRead        		: 2		: )
	                                		(BACnet_RemoteCycleTimeWrite   		: 1000	: )
	                                		(BACnet_RemoteFlagsWrite       		: 1		: )	*)
    _PresentValue_Priority12 AT%Q*: REAL;(* ~(BACnet_PresentValue_Priority12	:		: )	*)
	_StatusFlags AT%I*: WORD; 			(* ~(BACnet_StatusFlags 				:		: )	*)
	_StatusFlagsBits : ST_BACnet_StatusFlags;

	_nUpdateCount : UDINT := 0;
END_VAR
(* update client device *)
IF RemoteDevice._nUpdateCount = _nUpdateCount THEN
	RemoteDevice();
END_IF
(* remind current number of update counter *)
_nUpdateCount := RemoteDevice._nUpdateCount;

IF RemoteDevice.bFirstCycle THEN
	(* first call of the server device since reboot/reset *)
	bReady := FALSE;
	_PresentValue_Priority12 := F_BACnet_NAN();
ELSIF NOT RemoteDevice.bOperational THEN
	nErrorId := BACnet_ERR_OPERATIONAL;
	bReady := FALSE;

ELSIF _StatusFlags >= 4 THEN
	(* clear error flag *)
	nErrorId := BACnet_ERR_NO_ERROR;
	(* ready state *)
	bReady := TRUE;

	(* write into priority array *)
	IF bEnablePV THEN
		_PresentValue_Priority12	:= fPV;
	ELSE
		_PresentValue_Priority12	:= F_BACnet_NAN();
	END_IF

	(* present value *)
	fPresentValue := _PresentValue;

	(* build bit states *)
	_StatusFlagsBits := F_BACnet_StatusFlags(_StatusFlags);

	(* copy states to output *)
	bOverridden := _StatusFlagsBits.overridden;
	bOutOfService := _StatusFlagsBits.out_of_service;
	bFault := _StatusFlagsBits.fault;
	bInAlarm := _StatusFlagsBits.in_alarm;
ELSE
	(* server device not ready, reset local ready also *)
	bReady := FALSE;
	(* and set error ID *)
	nErrorId := BACnet_ERR_WRONG_MAPPING;
END_IF

(* set error flag *)
bError := (nErrorId <> BACnet_ERR_NO_ERROR);
END_FUNCTION_BLOCK

(* POU FB_BACnet_RemoteAnalogValue, ST *)
FUNCTION_BLOCK FB_BACnet_RemoteAnalogValue
VAR_INPUT
	bEnablePV		: BOOL; (* enable present value with priority x in priority array, FALSE = priority x disable *)
	fPV		: REAL; (* decimal number for priority x, when input bEnablePV is TRUE *)
END_VAR
VAR_IN_OUT
	RemoteDevice	: FB_BACnet_RemoteDevice;
END_VAR
VAR_OUTPUT
	bReady				: BOOL;
	fPresentValue		: REAL;
	bOverridden			: BOOL;
	bOutOfService		: BOOL;
	bFault				: BOOL;
	bInAlarm			: BOOL;
	bError				: BOOL;
	nErrorId			: UINT;
END_VAR
VAR
	_PresentValue AT%I*: REAL; 			(* ~(BACnet_PresentValue 				:		: )
								   			(BACnet_ObjectType 					: AV	: )
											(BACnet_RemoteCycletimeRead 		: 1000	: )
											(BACnet_RemoteFlagsRead        		: 1		: )
											(BACnet_RemoteResubscriptionInterval: 240	: )
	                                		(BACnet_RemoteCycleTimeWrite   		: 1000	: )
	                                		(BACnet_RemoteFlagsWrite       		: 1		: )	*)
    _PresentValue_Priority12 AT%Q*: REAL;(* ~(BACnet_PresentValue_Priority12	:		: )	*)
	_StatusFlags AT%I*: WORD; 			(* ~(BACnet_StatusFlags 				:		: )	*)
	_StatusFlagsBits : ST_BACnet_StatusFlags;

	_nUpdateCount : UDINT := 0;
END_VAR
(* update client device *)
IF RemoteDevice._nUpdateCount = _nUpdateCount THEN
	RemoteDevice();
END_IF
(* remind current number of update counter *)
_nUpdateCount := RemoteDevice._nUpdateCount;

IF RemoteDevice.bFirstCycle THEN
	(* first call of the server device since reboot/reset *)
	bReady := FALSE;
	_PresentValue_Priority12 := F_BACnet_NAN();
ELSIF NOT RemoteDevice.bOperational THEN
	nErrorId := BACnet_ERR_OPERATIONAL;
	bReady := FALSE;

ELSIF _StatusFlags >= 4 THEN
	(* clear error flag *)
	nErrorId := BACnet_ERR_NO_ERROR;
	(* ready state *)
	bReady := TRUE;

	(* write into priority array *)
	IF bEnablePV THEN
		_PresentValue_Priority12	:= fPV;
	ELSE
		_PresentValue_Priority12	:= F_BACnet_NAN();
	END_IF

	(* present value *)
	fPresentValue := _PresentValue;

	(* build bit states *)
	_StatusFlagsBits := F_BACnet_StatusFlags(_StatusFlags);

	(* copy states to output *)
	bOverridden := _StatusFlagsBits.overridden;
	bOutOfService := _StatusFlagsBits.out_of_service;
	bFault := _StatusFlagsBits.fault;
	bInAlarm := _StatusFlagsBits.in_alarm;
ELSE
	(* server device not ready, reset local ready also *)
	bReady := FALSE;
	(* and set error ID *)
	nErrorId := BACnet_ERR_WRONG_MAPPING;
END_IF

(* set error flag *)
bError := (nErrorId <> BACnet_ERR_NO_ERROR);
END_FUNCTION_BLOCK

(* POU FB_BACnet_RemoteAnalogValue_EX, ST *)
FUNCTION_BLOCK FB_BACnet_RemoteAnalogValue_EX
VAR_INPUT
	bEnablePV		: BOOL; (* enable present value with priority x in priority array, FALSE = priority x disable *)
	fPV		: REAL; (* decimal number for priority x, when input bEnablePV is TRUE *)
END_VAR
VAR_IN_OUT
	RemoteDevice	: FB_BACnet_RemoteDevice;
END_VAR
VAR_OUTPUT
	bReady				: BOOL;
	fPresentValue		: REAL;
	bOverridden			: BOOL;
	bOutOfService		: BOOL;
	bFault				: BOOL;
	bInAlarm			: BOOL;
	bOverRange			: BOOL;
	bUnderRange			: BOOL;
	bOtherFault			: BOOL;
	eEventState			: E_BACNETEVENTSTATE;
	tObjectID			: T_BACnet_ObjectIdentifier := 16#FFFFFFFF;
	bError				: BOOL;
	nErrorId			: UINT;
END_VAR
VAR
	_PresentValue AT%I*: REAL; 			(* ~(BACnet_PresentValue 				:		: )
								   			(BACnet_ObjectType 					: AV	: )
											(BACnet_RemoteCycletimeRead 		: 1000	: )
											(BACnet_RemoteFlagsRead        		: 1		: )
											(BACnet_RemoteResubscriptionInterval: 240	: )
	                                		(BACnet_RemoteCycleTimeWrite   		: 1000	: )
	                                		(BACnet_RemoteFlagsWrite       		: 1		: )	*)
    _PresentValue_Priority12 AT%Q*: REAL;(* ~(BACnet_PresentValue_Priority12	:		: )	*)
	_ObjectId AT%I*: DWORD;				(* ~(BACnet_ObjectIdentifier			:		: LINK) *)
	_StatusFlags AT%I*: WORD; 			(* ~(BACnet_StatusFlags 				:		: )	*)
	_Reliability AT%I*: WORD;			(* ~(BACnet_Reliability 				:		: )	*)
	_EventState AT%I*: WORD;			(* ~(BACnet_EventState					:		: )	*)
	_nUpdateCount : UDINT := 0;
	_StatusFlagsBits : ST_BACnet_StatusFlags;
END_VAR
(* update client device *)
IF RemoteDevice._nUpdateCount = _nUpdateCount THEN
	RemoteDevice();
END_IF
(* remind current number of update counter *)
_nUpdateCount := RemoteDevice._nUpdateCount;

IF RemoteDevice.bFirstCycle THEN
	(* first call of the server device since reboot/reset *)
	bReady := FALSE;
	_PresentValue_Priority12 := F_BACnet_NAN();
ELSIF NOT RemoteDevice.bOperational THEN
	nErrorId := BACnet_ERR_OPERATIONAL;
	bReady := FALSE;

ELSIF (F_BACnet_GetObjType(_ObjectId) <> BACnetObjectType_AnalogValue) THEN
	(* wrong mapping / invalid object ID *)
	IF _ObjectId = 0 THEN
		nErrorId := BACnet_ERR_WRONG_MAPPING;
	ELSE
		nErrorId := BACnet_ERR_INVALID_OBJECTID;
	END_IF
	bReady := FALSE;
	tObjectID := 16#FFFFFFFF;

ELSIF _StatusFlags >= 4 THEN
	(* clear error flag *)
	nErrorId := BACnet_ERR_NO_ERROR;
	(* ready state *)
	bReady := TRUE;

	(* write into priority array *)
	IF bEnablePV THEN
		_PresentValue_Priority12	:= fPV;
	ELSE
		_PresentValue_Priority12	:= F_BACnet_NAN();
	END_IF

	(* present value *)
	fPresentValue := _PresentValue;

	(* build bit states *)
	_StatusFlagsBits := F_BACnet_StatusFlags(_StatusFlags);

	(* copy states to output *)
	bOverridden := _StatusFlagsBits.overridden;
	bOutOfService := _StatusFlagsBits.out_of_service;
	bFault := _StatusFlagsBits.fault;
	bInAlarm := _StatusFlagsBits.in_alarm;
	bOverRange := (_Reliability = BACnetReliability_over_range);
	bUnderRange := (_Reliability = BACnetReliability_under_range);
	bOtherFault := (_Reliability = BACnetReliability_unreliable_other);
	eEventState := _EventState;
	tObjectID := _ObjectId;
ELSE
	(* server device not ready, reset local ready also *)
	bReady := FALSE;
	(* and set error ID *)
	nErrorId := BACnet_ERR_WRONG_MAPPING;
END_IF

(* set error flag *)
bError := (nErrorId <> BACnet_ERR_NO_ERROR);
END_FUNCTION_BLOCK

(* POU FB_BACnet_RemoteAnalogValue_POLL, ST *)
FUNCTION_BLOCK FB_BACnet_RemoteAnalogValue_POLL
VAR_INPUT
	bEnablePV		: BOOL; (* enable present value with priority x in priority array, FALSE = priority x disable *)
	fPV		: REAL; (* decimal number for priority x, when input bEnablePV is TRUE *)
END_VAR
VAR_IN_OUT
	RemoteDevice	: FB_BACnet_RemoteDevice;
END_VAR
VAR_OUTPUT
	bReady				: BOOL;
	fPresentValue		: REAL;
	bOverridden			: BOOL;
	bOutOfService		: BOOL;
	bFault				: BOOL;
	bInAlarm			: BOOL;
	bError				: BOOL;
	nErrorId			: UINT;
END_VAR
VAR
	_PresentValue AT%I*: REAL; 			(* ~(BACnet_PresentValue 				:		: )
								   			(BACnet_ObjectType 					: AV	: )
											(BACnet_RemoteCycletimeRead 		: 5000	: )
											(BACnet_RemoteFlagsRead        		: 2		: )
	                                		(BACnet_RemoteCycleTimeWrite   		: 1000	: )
	                                		(BACnet_RemoteFlagsWrite       		: 1		: )	*)
    _PresentValue_Priority12 AT%Q*: REAL;(* ~(BACnet_PresentValue_Priority12	:		: )	*)
	_StatusFlags AT%I*: WORD; 			(* ~(BACnet_StatusFlags 				:		: )	*)
	_StatusFlagsBits : ST_BACnet_StatusFlags;

	_nUpdateCount : UDINT := 0;
END_VAR
(* update client device *)
IF RemoteDevice._nUpdateCount = _nUpdateCount THEN
	RemoteDevice();
END_IF
(* remind current number of update counter *)
_nUpdateCount := RemoteDevice._nUpdateCount;

IF RemoteDevice.bFirstCycle THEN
	(* first call of the server device since reboot/reset *)
	bReady := FALSE;
	_PresentValue_Priority12 := F_BACnet_NAN();
ELSIF NOT RemoteDevice.bOperational THEN
	nErrorId := BACnet_ERR_OPERATIONAL;
	bReady := FALSE;

ELSIF _StatusFlags >= 4 THEN
	(* clear error flag *)
	nErrorId := BACnet_ERR_NO_ERROR;
	(* ready state *)
	bReady := TRUE;

	(* write into priority array *)
	IF bEnablePV THEN
		_PresentValue_Priority12	:= fPV;
	ELSE
		_PresentValue_Priority12	:= F_BACnet_NAN();
	END_IF

	(* present value *)
	fPresentValue := _PresentValue;

	(* build bit states *)
	_StatusFlagsBits := F_BACnet_StatusFlags(_StatusFlags);

	(* copy states to output *)
	bOverridden := _StatusFlagsBits.overridden;
	bOutOfService := _StatusFlagsBits.out_of_service;
	bFault := _StatusFlagsBits.fault;
	bInAlarm := _StatusFlagsBits.in_alarm;
ELSE
	(* server device not ready, reset local ready also *)
	bReady := FALSE;
	(* and set error ID *)
	nErrorId := BACnet_ERR_WRONG_MAPPING;
END_IF

(* set error flag *)
bError := (nErrorId <> BACnet_ERR_NO_ERROR);
END_FUNCTION_BLOCK

(* POU FB_BACnet_RemoteAveraging, ST *)
FUNCTION_BLOCK FB_BACnet_RemoteAveraging
VAR_IN_OUT
	RemoteDevice		: FB_BACnet_RemoteDevice;
END_VAR
VAR_OUTPUT
	bReady				: BOOL;
	nAverageValue		: REAL;
	bError				: BOOL;
	nErrorId			: UINT;
END_VAR
VAR
	_AverageValue AT%I*: REAL; 		(* ~(BACnet_AverageValue 				:		: )
										(BACnet_ObjectType					: AVG  	: )
										(BACnet_RemoteCycletimeRead 		: 1000	: )
										(BACnet_RemoteFlagsRead        		: 1		: )
										(BACnet_RemoteResubscriptionInterval: 240	: )
										(BACnet_RemoteCycleTimeWrite   		: 1000	: )
										(BACnet_RemoteFlagsWrite       		: 1		: )	*)

	_nUpdateCount : UDINT := 0;
END_VAR
(* update client device *)
IF RemoteDevice._nUpdateCount = _nUpdateCount THEN
	RemoteDevice();
END_IF
(* remind current number of update counter *)
_nUpdateCount := RemoteDevice._nUpdateCount;

IF RemoteDevice.bOperational THEN
	(* clear error flag *)
	nErrorId := BACnet_ERR_NO_ERROR;
	(* ready state *)
	bReady := TRUE;
	(* present value *)
	nAverageValue := _AverageValue;
ELSE
	(* server device not ready, reset local ready also *)
	bReady := FALSE;
	(* and set error ID *)
	nErrorId := BACnet_ERR_OPERATIONAL;
END_IF

(* set error flag *)
bError := (nErrorId <> BACnet_ERR_NO_ERROR);
END_FUNCTION_BLOCK

(* POU FB_BACnet_RemoteAveraging_EX, ST *)
FUNCTION_BLOCK FB_BACnet_RemoteAveraging_EX
VAR_IN_OUT
	RemoteDevice		: FB_BACnet_RemoteDevice;
END_VAR
VAR_OUTPUT
	bReady				: BOOL;
	nAverageValue		: REAL;
	tObjectID			: T_BACnet_ObjectIdentifier := 16#FFFFFFFF;
	bError				: BOOL;
	nErrorId			: UINT;
END_VAR
VAR
	_AverageValue AT%I*: REAL; 		(* ~(BACnet_AverageValue 				:		: )
										(BACnet_ObjectType					: AVG  	: )
										(BACnet_RemoteCycletimeRead 		: 1000	: )
										(BACnet_RemoteFlagsRead        		: 1		: )
										(BACnet_RemoteResubscriptionInterval: 240	: )
										(BACnet_RemoteCycleTimeWrite   		: 1000	: )
										(BACnet_RemoteFlagsWrite       		: 1		: )	*)
	_ObjectId AT%I*: DWORD;			(* ~(BACnet_ObjectIdentifier			:		: LINK) *)

	_nUpdateCount : UDINT := 0;
END_VAR
(* update client device *)
IF RemoteDevice._nUpdateCount = _nUpdateCount THEN
	RemoteDevice();
END_IF
(* remind current number of update counter *)
_nUpdateCount := RemoteDevice._nUpdateCount;

IF NOT RemoteDevice.bOperational THEN
	(* server device not ready, reset local ready also *)
	bReady := FALSE;
	(* and set error ID *)
	nErrorId := BACnet_ERR_OPERATIONAL;

ELSIF (F_BACnet_GetObjType(_ObjectId) <> BACnetObjectType_Averaging) THEN
	(* wrong mapping / invalid object ID *)
	IF _ObjectId = 0 THEN
		nErrorId := BACnet_ERR_WRONG_MAPPING;
	ELSE
		nErrorId := BACnet_ERR_INVALID_OBJECTID;
	END_IF
	bReady := FALSE;
	tObjectID := 16#FFFFFFFF;

ELSE
	(* clear error flag *)
	nErrorId := BACnet_ERR_NO_ERROR;
	(* ready state *)
	bReady := TRUE;
	(* present value *)
	nAverageValue := _AverageValue;
	tObjectID := _ObjectId;

END_IF

(* set error flag *)
bError := (nErrorId <> BACnet_ERR_NO_ERROR);
END_FUNCTION_BLOCK

(* POU FB_BACnet_RemoteAveraging_POLL, ST *)
FUNCTION_BLOCK FB_BACnet_RemoteAveraging_POLL
VAR_IN_OUT
	RemoteDevice		: FB_BACnet_RemoteDevice;
END_VAR
VAR_OUTPUT
	bReady				: BOOL;
	nAverageValue		: REAL;
	bError				: BOOL;
	nErrorId			: UINT;
END_VAR
VAR
	_AverageValue AT%I*: REAL; 		(* ~(BACnet_AverageValue 				:		: )
										(BACnet_ObjectType					: AVG  	: )
										(BACnet_RemoteCycletimeRead 		: 5000	: )
										(BACnet_RemoteFlagsRead        		: 2		: )
										(BACnet_RemoteCycleTimeWrite   		: 1000	: )
										(BACnet_RemoteFlagsWrite       		: 1		: )	*)

	_nUpdateCount : UDINT := 0;
END_VAR
(* update client device *)
IF RemoteDevice._nUpdateCount = _nUpdateCount THEN
	RemoteDevice();
END_IF
(* remind current number of update counter *)
_nUpdateCount := RemoteDevice._nUpdateCount;

IF RemoteDevice.bOperational THEN
	(* clear error flag *)
	nErrorId := BACnet_ERR_NO_ERROR;
	(* ready state *)
	bReady := TRUE;
	(* present value *)
	nAverageValue := _AverageValue;
ELSE
	(* server device not ready, reset local ready also *)
	bReady := FALSE;
	(* and set error ID *)
	nErrorId := BACnet_ERR_OPERATIONAL;
END_IF

(* set error flag *)
bError := (nErrorId <> BACnet_ERR_NO_ERROR);
END_FUNCTION_BLOCK

(* POU FB_BACnet_RemoteBinaryInput, ST *)
FUNCTION_BLOCK FB_BACnet_RemoteBinaryInput
VAR_OUTPUT
	bReady				: BOOL;
	bPresentValue		: BOOL;
	bOverridden			: BOOL;
	bOutOfService		: BOOL;
	bFault				: BOOL;
	bInAlarm			: BOOL;
	bError				: BOOL;
	nErrorId			: UINT;
END_VAR
VAR_IN_OUT
	RemoteDevice			: FB_BACnet_RemoteDevice;
END_VAR
VAR
	_PresentValue AT%I*: WORD; 				(* ~(BACnet_PresentValue 				:		: )
												(BACnet_ObjectType					: BI    : )
												(BACnet_RemoteCycletimeRead 		: 1000	: )
												(BACnet_RemoteFlagsRead        		: 1		: )
												(BACnet_RemoteResubscriptionInterval: 240	: )
		                                		(BACnet_RemoteCycleTimeWrite   		: 1000	: )
		                                		(BACnet_RemoteFlagsWrite       		: 1		: )	*)
	_StatusFlags AT%I*: WORD; 				(* ~(BACnet_StatusFlags 				:	    : )	*)
	_StatusFlagsBits : ST_BACnet_StatusFlags;
	_nUpdateCount : UDINT := 0;
END_VAR
(* update client device *)
IF RemoteDevice._nUpdateCount = _nUpdateCount THEN
	RemoteDevice();
END_IF
(* remind current number of update counter *)
_nUpdateCount := RemoteDevice._nUpdateCount;

IF NOT RemoteDevice.bOperational THEN
	nErrorId := BACnet_ERR_OPERATIONAL;
	bReady := FALSE;

ELSIF _StatusFlags >= 4 THEN
	(* clear error flag *)
	nErrorId := BACnet_ERR_NO_ERROR;
	(* ready state *)
	bReady := TRUE;

	(* present value *)
	bPresentValue := F_BinPV_To_Bool(_PresentValue);

	(* build bit states *)
	_StatusFlagsBits := F_BACnet_StatusFlags(_StatusFlags);

	(* copy states to output *)
	bOverridden := _StatusFlagsBits.overridden;
	bOutOfService := _StatusFlagsBits.out_of_service;
	bFault := _StatusFlagsBits.fault;
	bInAlarm := _StatusFlagsBits.in_alarm;

ELSE
	bReady := FALSE;
	(* and set error ID *)
	nErrorId := BACnet_ERR_WRONG_MAPPING;
END_IF

(* set error flag *)
bError := (nErrorId <> BACnet_ERR_NO_ERROR);
END_FUNCTION_BLOCK

(* POU FB_BACnet_RemoteBinaryInput_EX, ST *)
FUNCTION_BLOCK FB_BACnet_RemoteBinaryInput_EX
VAR_OUTPUT
	bReady				: BOOL;
	bPresentValue		: BOOL;
	bOverridden			: BOOL;
	bOutOfService		: BOOL;
	bFault				: BOOL;
	bInAlarm			: BOOL;
	bNoSensor			: BOOL;
	bOpenLoop			: BOOL;
	bShortedLoop		: BOOL;
	bOtherFault			: BOOL;
	eEventState			: E_BACNETEVENTSTATE;
	nChangeOfState		: UDINT;
	tObjectID			: T_BACnet_ObjectIdentifier := 16#FFFFFFFF;
	bError				: BOOL;
	nErrorId			: UINT;
END_VAR
VAR_IN_OUT
	RemoteDevice			: FB_BACnet_RemoteDevice;
END_VAR
VAR
	_ChangeOfStateCount AT%I*: UDINT;	(* ~(BACnet_ChangeOfStateCount			:		: ) *)
	_ObjectId AT%I*: DWORD;				(* ~(BACnet_ObjectIdentifier			:		: LINK) *)
	_PresentValue AT%I*: WORD; 			(* ~(BACnet_PresentValue 				:		: )
											(BACnet_ObjectType					: BI    : )
											(BACnet_RemoteCycletimeRead 		: 1000	: )
											(BACnet_RemoteFlagsRead        		: 1		: )
											(BACnet_RemoteResubscriptionInterval: 240	: )
		                                	(BACnet_RemoteCycleTimeWrite   		: 1000	: )
		                                	(BACnet_RemoteFlagsWrite       		: 1		: )	*)
	_StatusFlags AT%I*: WORD; 			(* ~(BACnet_StatusFlags 				:	    : )	*)
	_Reliability AT%I*: WORD; 			(* ~(BACnet_Reliability 				:		: )	*)
	_EventState AT%I*: WORD;			(* ~(BACnet_EventState					:		: )	*)
	_nUpdateCount : UDINT := 0;
	_StatusFlagsBits : ST_BACnet_StatusFlags;
END_VAR
(* update client device *)
IF RemoteDevice._nUpdateCount = _nUpdateCount THEN
	RemoteDevice();
END_IF
(* remind current number of update counter *)
_nUpdateCount := RemoteDevice._nUpdateCount;

IF NOT RemoteDevice.bOperational THEN
	nErrorId := BACnet_ERR_OPERATIONAL;
	bReady := FALSE;

ELSIF (F_BACnet_GetObjType(_ObjectId) <> BACnetObjectType_BinaryInput) THEN
	(* wrong mapping / invalid object ID *)
	IF _ObjectId = 0 THEN
		nErrorId := BACnet_ERR_WRONG_MAPPING;
	ELSE
		nErrorId := BACnet_ERR_INVALID_OBJECTID;
	END_IF
	bReady := FALSE;
	tObjectID := 16#FFFFFFFF;

ELSIF _StatusFlags >= 4 THEN
	(* clear error flag *)
	nErrorId := BACnet_ERR_NO_ERROR;
	(* ready state *)
	bReady := TRUE;

	(* present value *)
	bPresentValue := F_BinPV_To_Bool(_PresentValue);

	(* build bit states *)
	_StatusFlagsBits := F_BACnet_StatusFlags(_StatusFlags);

	(* copy states to output *)
	bOverridden := _StatusFlagsBits.overridden;
	bOutOfService := _StatusFlagsBits.out_of_service;
	bFault := _StatusFlagsBits.fault;
	bInAlarm := _StatusFlagsBits.in_alarm;
	bNoSensor := (_Reliability = BACnetReliability_no_sensor);
	bOpenLoop := (_Reliability = BACnetReliability_open_loop);
	bShortedLoop := (_Reliability = BACnetReliability_shorted_loop);
	bOtherFault := (_Reliability = BACnetReliability_unreliable_other);
	eEventState := _EventState;
	tObjectID := _ObjectId;

	(* copy change_of_state_count *)
	nChangeOfState := _ChangeOfStateCount;

ELSE
	bReady := FALSE;
	(* and set error ID *)
	nErrorId := BACnet_ERR_WRONG_MAPPING;
END_IF

(* set error flag *)
bError := (nErrorId <> BACnet_ERR_NO_ERROR);
END_FUNCTION_BLOCK

(* POU FB_BACnet_RemoteBinaryInput_POLL, ST *)
FUNCTION_BLOCK FB_BACnet_RemoteBinaryInput_POLL
VAR_OUTPUT
	bReady				: BOOL;
	bPresentValue		: BOOL;
	bOverridden			: BOOL;
	bOutOfService		: BOOL;
	bFault				: BOOL;
	bInAlarm			: BOOL;
	bError				: BOOL;
	nErrorId			: UINT;
END_VAR
VAR_IN_OUT
	RemoteDevice			: FB_BACnet_RemoteDevice;
END_VAR
VAR
	_PresentValue AT%I*: WORD; 				(* ~(BACnet_PresentValue 				:		: )
												(BACnet_ObjectType					: BI    : )
												(BACnet_RemoteCycletimeRead 		: 5000	: )
												(BACnet_RemoteFlagsRead        		: 2		: )
		                                		(BACnet_RemoteCycleTimeWrite   		: 1000	: )
		                                		(BACnet_RemoteFlagsWrite       		: 1		: )	*)
	_StatusFlags AT%I*: WORD; 				(* ~(BACnet_StatusFlags 				:	    : )	*)
	_StatusFlagsBits : ST_BACnet_StatusFlags;
	_nUpdateCount : UDINT := 0;
END_VAR
(* update client device *)
IF RemoteDevice._nUpdateCount = _nUpdateCount THEN
	RemoteDevice();
END_IF
(* remind current number of update counter *)
_nUpdateCount := RemoteDevice._nUpdateCount;

IF NOT RemoteDevice.bOperational THEN
	nErrorId := BACnet_ERR_OPERATIONAL;
	bReady := FALSE;

ELSIF _StatusFlags >= 4 THEN
	(* clear error flag *)
	nErrorId := BACnet_ERR_NO_ERROR;
	(* ready state *)
	bReady := TRUE;

	(* present value *)
	bPresentValue := F_BinPV_To_Bool(_PresentValue);

	(* build bit states *)
	_StatusFlagsBits := F_BACnet_StatusFlags(_StatusFlags);

	(* copy states to output *)
	bOverridden := _StatusFlagsBits.overridden;
	bOutOfService := _StatusFlagsBits.out_of_service;
	bFault := _StatusFlagsBits.fault;
	bInAlarm := _StatusFlagsBits.in_alarm;

ELSE
	bReady := FALSE;
	(* and set error ID *)
	nErrorId := BACnet_ERR_WRONG_MAPPING;
END_IF

(* set error flag *)
bError := (nErrorId <> BACnet_ERR_NO_ERROR);
END_FUNCTION_BLOCK

(* POU FB_BACnet_RemoteBinaryOutput, ST *)
FUNCTION_BLOCK FB_BACnet_RemoteBinaryOutput
VAR_INPUT
	bEnablePV	: BOOL; (* enable present value with priority x in priority array, FALSE = priority x disable (NULL) *)
	bPV			: BOOL; (* present value bool type *)
END_VAR
VAR_IN_OUT
	RemoteDevice	: FB_BACnet_RemoteDevice;
END_VAR
VAR_OUTPUT
	bReady				: BOOL;
	bPresentValue		: BOOL;
	bOverridden			: BOOL;
	bOutOfService		: BOOL;
	bFault				: BOOL;
	bInAlarm			: BOOL;
	bError				: BOOL;
	nErrorId			: UINT;
END_VAR
VAR
	_PresentValue AT%I*: WORD; 			(* ~(BACnet_PresentValue 				:		: )
								   			(BACnet_ObjectType 					: BO	: )
											(BACnet_RemoteCycletimeRead 		: 1000	: )
											(BACnet_RemoteFlagsRead        		: 1		: )
											(BACnet_RemoteResubscriptionInterval: 240	: )
		                            		(BACnet_RemoteCycleTimeWrite   		: 1000	: )
		                            		(BACnet_RemoteFlagsWrite       		: 1		: )	*)
    _PresentValue_Priority12 AT%Q*: WORD;(* ~(BACnet_PresentValue_Priority12	:		: )	*)
	_StatusFlags AT%I*: WORD; 			(* ~(BACnet_StatusFlags 				:		: )	*)
	_StatusFlagsBits : ST_BACnet_StatusFlags;
	_nUpdateCount : UDINT := 0;
END_VAR
(* update client device *)
IF RemoteDevice._nUpdateCount = _nUpdateCount THEN
	RemoteDevice();
END_IF
(* remind current number of update counter *)
_nUpdateCount := RemoteDevice._nUpdateCount;

IF RemoteDevice.bFirstCycle THEN
	(* first call of the server device since reboot/reset *)
	bReady := FALSE;
	_PresentValue_Priority12 := BACnetBinaryPV_NULL;
ELSIF NOT RemoteDevice.bOperational THEN
	nErrorId := BACnet_ERR_OPERATIONAL;
	bReady := FALSE;

ELSIF _StatusFlags >= 4 THEN
	(* clear error flag *)
	nErrorId := BACnet_ERR_NO_ERROR;
	(* ready state *)
	bReady := TRUE;

	(* write into priority array *)
	_PresentValue_Priority12 := F_Bool_To_BinPV(bEnablePV, bPV);

	(* present value *)
	bPresentValue := F_BinPV_To_Bool(_PresentValue);

	(* build bit states *)
	_StatusFlagsBits := F_BACnet_StatusFlags(_StatusFlags);

	(* copy states to output *)
	bOverridden := _StatusFlagsBits.overridden;
	bOutOfService := _StatusFlagsBits.out_of_service;
	bFault := _StatusFlagsBits.fault;
	bInAlarm := _StatusFlagsBits.in_alarm;
ELSE
	(* server device not ready, reset local ready also *)
	bReady := FALSE;
	(* and set error ID *)
	nErrorId := BACnet_ERR_WRONG_MAPPING;
END_IF

(* set error flag *)
bError := (nErrorId <> BACnet_ERR_NO_ERROR);
END_FUNCTION_BLOCK

(* POU FB_BACnet_RemoteBinaryOutput_EX, ST *)
FUNCTION_BLOCK FB_BACnet_RemoteBinaryOutput_EX
VAR_INPUT
	bEnablePV	: BOOL; (* enable present value with priority x in priority array, FALSE = priority x disable (NULL) *)
	bPV			: BOOL; (* present value bool type *)
END_VAR
VAR_IN_OUT
	RemoteDevice	: FB_BACnet_RemoteDevice;
END_VAR
VAR_OUTPUT
	bReady				: BOOL;
	bPresentValue		: BOOL;
	bOverridden			: BOOL;
	bOutOfService		: BOOL;
	bFault				: BOOL;
	bInAlarm			: BOOL;
	bNoOutput			: BOOL;
	bOpenLoop			: BOOL;
	bShortedLoop		: BOOL;
	bOtherFault			: BOOL;
	eEventState			: E_BACNETEVENTSTATE;
	nChangeOfState		: UDINT;
	tObjectID			: T_BACnet_ObjectIdentifier := 16#FFFFFFFF;
	bError				: BOOL;
	nErrorId			: UINT;
END_VAR
VAR
	_ChangeOfStateCount AT%I*: UDINT;	(* ~(BACnet_ChangeOfStateCount			:		: ) *)
	_ObjectId AT%I*: DWORD;				(* ~(BACnet_ObjectIdentifier			:		: LINK) *)
	_PresentValue AT%I*: WORD; 			(* ~(BACnet_PresentValue 				:		: )
								   			(BACnet_ObjectType 					: BO	: )
											(BACnet_RemoteCycletimeRead 		: 1000	: )
											(BACnet_RemoteFlagsRead        		: 1		: )
											(BACnet_RemoteResubscriptionInterval: 240	: )
		                            		(BACnet_RemoteCycleTimeWrite   		: 1000	: )
		                            		(BACnet_RemoteFlagsWrite       		: 1		: )	*)
	_StatusFlags AT%I*: WORD; 			(* ~(BACnet_StatusFlags 				:		: )	*)
	_Reliability AT%I*: WORD;			(* ~(BACnet_Reliability 				:		: )	*)
	_EventState AT%I*: WORD;			(* ~(BACnet_EventState					:		: )	*)
    _PresentValue_Priority12 AT%Q*: WORD;(* ~(BACnet_PresentValue_Priority12	:		: )	*)
	_nUpdateCount : UDINT := 0;
	_StatusFlagsBits : ST_BACnet_StatusFlags;
END_VAR
(* update client device *)
IF RemoteDevice._nUpdateCount = _nUpdateCount THEN
	RemoteDevice();
END_IF
(* remind current number of update counter *)
_nUpdateCount := RemoteDevice._nUpdateCount;

IF RemoteDevice.bFirstCycle THEN
	(* first call of the server device since reboot/reset *)
	bReady := FALSE;
	_PresentValue_Priority12 := BACnetBinaryPV_NULL;
ELSIF NOT RemoteDevice.bOperational THEN
	nErrorId := BACnet_ERR_OPERATIONAL;
	bReady := FALSE;

ELSIF (F_BACnet_GetObjType(_ObjectId) <> BACnetObjectType_BinaryOutput) THEN
	(* wrong mapping / invalid object ID *)
	IF _ObjectId = 0 THEN
		nErrorId := BACnet_ERR_WRONG_MAPPING;
	ELSE
		nErrorId := BACnet_ERR_INVALID_OBJECTID;
	END_IF
	bReady := FALSE;
	tObjectID := 16#FFFFFFFF;

ELSIF _StatusFlags >= 4 THEN
	(* clear error flag *)
	nErrorId := BACnet_ERR_NO_ERROR;
	(* ready state *)
	bReady := TRUE;

	(* write into priority array *)
	_PresentValue_Priority12 := F_Bool_To_BinPV(bEnablePV, bPV);

	(* present value *)
	bPresentValue := F_BinPV_To_Bool(_PresentValue);

	(* build bit states *)
	_StatusFlagsBits := F_BACnet_StatusFlags(_StatusFlags);

	(* copy states to output *)
	bOverridden := _StatusFlagsBits.overridden;
	bOutOfService := _StatusFlagsBits.out_of_service;
	bFault := _StatusFlagsBits.fault;
	bInAlarm := _StatusFlagsBits.in_alarm;
	bNoOutput := (_Reliability = BACnetReliability_no_output);
	bOpenLoop := (_Reliability = BACnetReliability_open_loop);
	bShortedLoop := (_Reliability = BACnetReliability_shorted_loop);
	bOtherFault := (_Reliability = BACnetReliability_unreliable_other);
	eEventState := _EventState;
	tObjectID := _ObjectId;

	(* copy change_of_state_count *)
	nChangeOfState := _ChangeOfStateCount;
ELSE
	(* server device not ready, reset local ready also *)
	bReady := FALSE;
	(* and set error ID *)
	nErrorId := BACnet_ERR_WRONG_MAPPING;
END_IF

(* set error flag *)
bError := (nErrorId <> BACnet_ERR_NO_ERROR);
END_FUNCTION_BLOCK

(* POU FB_BACnet_RemoteBinaryOutput_POLL, ST *)
FUNCTION_BLOCK FB_BACnet_RemoteBinaryOutput_POLL
VAR_INPUT
	bEnablePV	: BOOL; (* enable present value with priority x in priority array, FALSE = priority x disable (NULL) *)
	bPV			: BOOL; (* present value bool type *)
END_VAR
VAR_IN_OUT
	RemoteDevice	: FB_BACnet_RemoteDevice;
END_VAR
VAR_OUTPUT
	bReady				: BOOL;
	bPresentValue		: BOOL;
	bOverridden			: BOOL;
	bOutOfService		: BOOL;
	bFault				: BOOL;
	bInAlarm			: BOOL;
	bError				: BOOL;
	nErrorId			: UINT;
END_VAR
VAR
	_PresentValue AT%I*: WORD; 			(* ~(BACnet_PresentValue 				:		: )
								   			(BACnet_ObjectType 					: BO	: )
											(BACnet_RemoteCycletimeRead 		: 5000	: )
											(BACnet_RemoteFlagsRead        		: 2		: )
		                            		(BACnet_RemoteCycleTimeWrite   		: 1000	: )
		                            		(BACnet_RemoteFlagsWrite       		: 1		: )	*)
    _PresentValue_Priority12 AT%Q*: WORD;(* ~(BACnet_PresentValue_Priority12	:		: )	*)
	_StatusFlags AT%I*: WORD; 			(* ~(BACnet_StatusFlags 				:		: )	*)
	_StatusFlagsBits : ST_BACnet_StatusFlags;
	_nUpdateCount : UDINT := 0;
END_VAR
(* update client device *)
IF RemoteDevice._nUpdateCount = _nUpdateCount THEN
	RemoteDevice();
END_IF
(* remind current number of update counter *)
_nUpdateCount := RemoteDevice._nUpdateCount;

IF RemoteDevice.bFirstCycle THEN
	(* first call of the server device since reboot/reset *)
	bReady := FALSE;
	_PresentValue_Priority12 := BACnetBinaryPV_NULL;
ELSIF NOT RemoteDevice.bOperational THEN
	nErrorId := BACnet_ERR_OPERATIONAL;
	bReady := FALSE;

ELSIF _StatusFlags >= 4 THEN
	(* clear error flag *)
	nErrorId := BACnet_ERR_NO_ERROR;
	(* ready state *)
	bReady := TRUE;

	(* write into priority array *)
	_PresentValue_Priority12 := F_Bool_To_BinPV(bEnablePV, bPV);

	(* present value *)
	bPresentValue := F_BinPV_To_Bool(_PresentValue);

	(* build bit states *)
	_StatusFlagsBits := F_BACnet_StatusFlags(_StatusFlags);

	(* copy states to output *)
	bOverridden := _StatusFlagsBits.overridden;
	bOutOfService := _StatusFlagsBits.out_of_service;
	bFault := _StatusFlagsBits.fault;
	bInAlarm := _StatusFlagsBits.in_alarm;
ELSE
	(* server device not ready, reset local ready also *)
	bReady := FALSE;
	(* and set error ID *)
	nErrorId := BACnet_ERR_WRONG_MAPPING;
END_IF

(* set error flag *)
bError := (nErrorId <> BACnet_ERR_NO_ERROR);
END_FUNCTION_BLOCK

(* POU FB_BACnet_RemoteBinaryValue, ST *)
FUNCTION_BLOCK FB_BACnet_RemoteBinaryValue
VAR_INPUT
	bEnablePV	: BOOL; (* enable present value with priority x in priority array, FALSE = priority x disable (NULL) *)
	bPV			: BOOL; (* present value bool type *)
END_VAR
VAR_IN_OUT
	RemoteDevice		: FB_BACnet_RemoteDevice;
END_VAR
VAR_OUTPUT
	bReady				: BOOL;
	bPresentValue		: BOOL;
	bOverridden			: BOOL;
	bOutOfService		: BOOL;
	bFault				: BOOL;
	bInAlarm			: BOOL;
	bError				: BOOL;
	nErrorId			: UINT;
END_VAR
VAR

	_PresentValue AT%I*: WORD; 			(* ~(BACnet_PresentValue 				:		: )
								   			(BACnet_ObjectType 					: BV	: )
											(BACnet_RemoteCycletimeRead 		: 1000	: )
											(BACnet_RemoteFlagsRead        		: 1		: )
											(BACnet_RemoteResubscriptionInterval: 240	: )
	                                		(BACnet_RemoteCycleTimeWrite   		: 1000	: )
	                                		(BACnet_RemoteFlagsWrite       		: 1		: )	*)
    _PresentValue_Priority12 AT%Q*: WORD;(* ~(BACnet_PresentValue_Priority12	:		: )	*)
	_StatusFlags AT%I*: WORD; 			(* ~(BACnet_StatusFlags 				:		: )	*)
	_StatusFlagsBits : ST_BACnet_StatusFlags;

	_nUpdateCount : UDINT := 0;
END_VAR
(* update client device *)
IF RemoteDevice._nUpdateCount = _nUpdateCount THEN
	RemoteDevice();
END_IF
(* remind current number of update counter *)
_nUpdateCount := RemoteDevice._nUpdateCount;

IF RemoteDevice.bFirstCycle THEN
	(* first call of the server device since reboot/reset *)
	bReady := FALSE;
	_PresentValue_Priority12 := BACnetBinaryPV_NULL;
ELSIF NOT RemoteDevice.bOperational THEN
	nErrorId := BACnet_ERR_OPERATIONAL;
	bReady := FALSE;

ELSIF _StatusFlags >= 4 THEN
	(* clear error flag *)
	nErrorId := BACnet_ERR_NO_ERROR;
	(* ready state *)
	bReady := TRUE;

	(* write into priority array *)
	_PresentValue_Priority12 := F_Bool_To_BinPV(bEnablePV, bPV);

	(* present value *)
	bPresentValue := F_BinPV_To_Bool(_PresentValue);

	(* build bit states *)
	_StatusFlagsBits := F_BACnet_StatusFlags(_StatusFlags);

	(* copy states to output *)
	bOverridden := _StatusFlagsBits.overridden;
	bOutOfService := _StatusFlagsBits.out_of_service;
	bFault := _StatusFlagsBits.fault;
	bInAlarm := _StatusFlagsBits.in_alarm;

ELSE
	(* server device not ready, reset local ready also *)
	bReady := FALSE;
	(* and set error ID *)
	nErrorId := BACnet_ERR_WRONG_MAPPING;
END_IF

(* set error flag *)
bError := (nErrorId <> BACnet_ERR_NO_ERROR);
END_FUNCTION_BLOCK

(* POU FB_BACnet_RemoteBinaryValue_EX, ST *)
FUNCTION_BLOCK FB_BACnet_RemoteBinaryValue_EX
VAR_INPUT
	bEnablePV	: BOOL; (* enable present value with priority x in priority array, FALSE = priority x disable (NULL) *)
	bPV			: BOOL; (* present value bool type *)
END_VAR
VAR_IN_OUT
	RemoteDevice		: FB_BACnet_RemoteDevice;
END_VAR
VAR_OUTPUT
	bReady				: BOOL;
	bPresentValue		: BOOL;
	bOverridden			: BOOL;
	bOutOfService		: BOOL;
	bFault				: BOOL;
	bInAlarm			: BOOL;
	bOtherFault			: BOOL;
	eEventState			: E_BACNETEVENTSTATE;
	nChangeOfState		: UDINT;
	tObjectID			: T_BACnet_ObjectIdentifier := 16#FFFFFFFF;
	bError				: BOOL;
	nErrorId			: UINT;
END_VAR
VAR
	_ChangeOfStateCount AT%I*: UDINT;	(* ~(BACnet_ChangeOfStateCount			:		: ) *)
	_ObjectId AT%I*: DWORD;				(* ~(BACnet_ObjectIdentifier			:		: LINK) *)
	_PresentValue AT%I*: WORD; 			(* ~(BACnet_PresentValue 				:		: )
								   			(BACnet_ObjectType 					: BV	: )
											(BACnet_RemoteCycletimeRead 		: 1000	: )
											(BACnet_RemoteFlagsRead        		: 1		: )
											(BACnet_RemoteResubscriptionInterval: 240	: )
	                                		(BACnet_RemoteCycleTimeWrite   		: 1000	: )
	                                		(BACnet_RemoteFlagsWrite       		: 1		: )	*)
	_StatusFlags AT%I*: WORD; 			(* ~(BACnet_StatusFlags 				:		: )	*)
	_Reliability AT%I*: WORD;			(* ~(BACnet_Reliability 				:		: )	*)
	_EventState AT%I*: WORD;			(* ~(BACnet_EventState					:		: )	*)
    _PresentValue_Priority12 AT%Q*: WORD;(* ~(BACnet_PresentValue_Priority12	:		: )	*)
	_nUpdateCount : UDINT := 0;
	_StatusFlagsBits : ST_BACnet_StatusFlags;
END_VAR
(* update client device *)
IF RemoteDevice._nUpdateCount = _nUpdateCount THEN
	RemoteDevice();
END_IF
(* remind current number of update counter *)
_nUpdateCount := RemoteDevice._nUpdateCount;

IF RemoteDevice.bFirstCycle THEN
	(* first call of the server device since reboot/reset *)
	bReady := FALSE;
	_PresentValue_Priority12 := BACnetBinaryPV_NULL;
ELSIF NOT RemoteDevice.bOperational THEN
	nErrorId := BACnet_ERR_OPERATIONAL;
	bReady := FALSE;

ELSIF (F_BACnet_GetObjType(_ObjectId) <> BACnetObjectType_BinaryValue) THEN
	(* wrong mapping / invalid object ID *)
	IF _ObjectId = 0 THEN
		nErrorId := BACnet_ERR_WRONG_MAPPING;
	ELSE
		nErrorId := BACnet_ERR_INVALID_OBJECTID;
	END_IF
	bReady := FALSE;
	tObjectID := 16#FFFFFFFF;

ELSIF _StatusFlags >= 4 THEN
	(* clear error flag *)
	nErrorId := BACnet_ERR_NO_ERROR;
	(* ready state *)
	bReady := TRUE;

	(* write into priority array *)
	_PresentValue_Priority12 := F_Bool_To_BinPV(bEnablePV, bPV);

	(* present value *)
	bPresentValue := F_BinPV_To_Bool(_PresentValue);

	(* build bit states *)
	_StatusFlagsBits := F_BACnet_StatusFlags(_StatusFlags);

	(* copy states to output *)
	bOverridden := _StatusFlagsBits.overridden;
	bOutOfService := _StatusFlagsBits.out_of_service;
	bFault := _StatusFlagsBits.fault;
	bInAlarm := _StatusFlagsBits.in_alarm;
	bOtherFault := (_Reliability = BACnetReliability_unreliable_other);
	eEventState := _EventState;
	tObjectID := _ObjectId;

	(* copy change_of_state_count *)
	nChangeOfState := _ChangeOfStateCount;

ELSE
	(* server device not ready, reset local ready also *)
	bReady := FALSE;
	(* and set error ID *)
	nErrorId := BACnet_ERR_WRONG_MAPPING;
END_IF

(* set error flag *)
bError := (nErrorId <> BACnet_ERR_NO_ERROR);
END_FUNCTION_BLOCK

(* POU FB_BACnet_RemoteBinaryValue_POLL, ST *)
FUNCTION_BLOCK FB_BACnet_RemoteBinaryValue_POLL
VAR_INPUT
	bEnablePV	: BOOL; (* enable present value with priority x in priority array, FALSE = priority x disable (NULL) *)
	bPV			: BOOL; (* present value bool type *)
END_VAR
VAR_IN_OUT
	RemoteDevice		: FB_BACnet_RemoteDevice;
END_VAR
VAR_OUTPUT
	bReady				: BOOL;
	bPresentValue		: BOOL;
	bOverridden			: BOOL;
	bOutOfService		: BOOL;
	bFault				: BOOL;
	bInAlarm			: BOOL;
	bError				: BOOL;
	nErrorId			: UINT;
END_VAR
VAR

	_PresentValue AT%I*: WORD; 			(* ~(BACnet_PresentValue 				:		: )
								   			(BACnet_ObjectType 					: BV	: )
											(BACnet_RemoteCycletimeRead 		: 5000	: )
											(BACnet_RemoteFlagsRead        		: 2		: )
	                                		(BACnet_RemoteCycleTimeWrite   		: 1000	: )
	                                		(BACnet_RemoteFlagsWrite       		: 1		: )	*)
    _PresentValue_Priority12 AT%Q*: WORD;(* ~(BACnet_PresentValue_Priority12	:		: )	*)
	_StatusFlags AT%I*: WORD; 			(* ~(BACnet_StatusFlags 				:		: )	*)
	_StatusFlagsBits : ST_BACnet_StatusFlags;

	_nUpdateCount : UDINT := 0;
END_VAR
(* update client device *)
IF RemoteDevice._nUpdateCount = _nUpdateCount THEN
	RemoteDevice();
END_IF
(* remind current number of update counter *)
_nUpdateCount := RemoteDevice._nUpdateCount;

IF RemoteDevice.bFirstCycle THEN
	(* first call of the server device since reboot/reset *)
	bReady := FALSE;
	_PresentValue_Priority12 := BACnetBinaryPV_NULL;
ELSIF NOT RemoteDevice.bOperational THEN
	nErrorId := BACnet_ERR_OPERATIONAL;
	bReady := FALSE;

ELSIF _StatusFlags >= 4 THEN
	(* clear error flag *)
	nErrorId := BACnet_ERR_NO_ERROR;
	(* ready state *)
	bReady := TRUE;

	(* write into priority array *)
	_PresentValue_Priority12 := F_Bool_To_BinPV(bEnablePV, bPV);

	(* present value *)
	bPresentValue := F_BinPV_To_Bool(_PresentValue);

	(* build bit states *)
	_StatusFlagsBits := F_BACnet_StatusFlags(_StatusFlags);

	(* copy states to output *)
	bOverridden := _StatusFlagsBits.overridden;
	bOutOfService := _StatusFlagsBits.out_of_service;
	bFault := _StatusFlagsBits.fault;
	bInAlarm := _StatusFlagsBits.in_alarm;

ELSE
	(* server device not ready, reset local ready also *)
	bReady := FALSE;
	(* and set error ID *)
	nErrorId := BACnet_ERR_WRONG_MAPPING;
END_IF

(* set error flag *)
bError := (nErrorId <> BACnet_ERR_NO_ERROR);
END_FUNCTION_BLOCK

(* POU FB_BACnet_RemoteCalendar, ST *)
FUNCTION_BLOCK FB_BACnet_RemoteCalendar
VAR_IN_OUT
	RemoteDevice		: FB_BACnet_RemoteDevice;
END_VAR
VAR_OUTPUT
	bReady				: BOOL;
	bPresentValue		: BOOL;
	bError				: BOOL;
	nErrorId			: UINT;
END_VAR
VAR
	_PresentValue AT%I*: BOOL;	(* ~(BACnet_PresentValue 				:		: )
									(BACnet_ObjectType 					: CAL	: )
									(BACnet_RemoteCycletimeRead 		: 1000	: )
									(BACnet_RemoteFlagsRead        		: 1		: )
									(BACnet_RemoteResubscriptionInterval: 240	: )
                            		(BACnet_RemoteCycleTimeWrite   		: 1000	: )
                            		(BACnet_RemoteFlagsWrite       		: 1		: )	*)
	_nUpdateCount : UDINT := 0;
END_VAR
(* update client device *)
IF RemoteDevice._nUpdateCount = _nUpdateCount THEN
	RemoteDevice();
END_IF
(* remind current number of update counter *)
_nUpdateCount := RemoteDevice._nUpdateCount;

IF RemoteDevice.bOperational THEN
	(* clear error flag *)
	nErrorId := BACnet_ERR_NO_ERROR;
	(* ready state *)
	bReady := TRUE;
	(* present value *)
	bPresentValue := _PresentValue;
ELSE
	(* server device not ready, reset local ready also *)
	bReady := FALSE;
	(* and set error ID *)
	nErrorId := BACnet_ERR_OPERATIONAL;
END_IF

(* set error flag *)
bError := (nErrorId <> BACnet_ERR_NO_ERROR);
END_FUNCTION_BLOCK

(* POU FB_BACnet_RemoteCalendar_EX, ST *)
FUNCTION_BLOCK FB_BACnet_RemoteCalendar_EX
VAR_IN_OUT
	RemoteDevice		: FB_BACnet_RemoteDevice;
END_VAR
VAR_OUTPUT
	bReady				: BOOL;
	bPresentValue		: BOOL;
	tObjectID			: T_BACnet_ObjectIdentifier := 16#FFFFFFFF;
	bError				: BOOL;
	nErrorId			: UINT;
END_VAR
VAR
	_PresentValue AT%I*: BOOL;	(* ~(BACnet_PresentValue 				:		: )
									(BACnet_ObjectType 					: CAL	: )
									(BACnet_RemoteCycletimeRead 		: 1000	: )
									(BACnet_RemoteFlagsRead        		: 1		: )
									(BACnet_RemoteResubscriptionInterval: 240	: )
                            		(BACnet_RemoteCycleTimeWrite   		: 1000	: )
                            		(BACnet_RemoteFlagsWrite       		: 1		: )	*)
	_ObjectId AT%I*: DWORD;		(* ~(BACnet_ObjectIdentifier			:		: LINK) *)
	_nUpdateCount : UDINT := 0;
END_VAR
(* update client device *)
IF RemoteDevice._nUpdateCount = _nUpdateCount THEN
	RemoteDevice();
END_IF
(* remind current number of update counter *)
_nUpdateCount := RemoteDevice._nUpdateCount;

IF NOT RemoteDevice.bOperational THEN
	nErrorId := BACnet_ERR_OPERATIONAL;
	bReady := FALSE;

ELSIF (F_BACnet_GetObjType(_ObjectId) <> BACnetObjectType_Calendar) THEN
	(* wrong mapping / invalid object ID *)
	IF _ObjectId = 0 THEN
		nErrorId := BACnet_ERR_WRONG_MAPPING;
	ELSE
		nErrorId := BACnet_ERR_INVALID_OBJECTID;
	END_IF
	bReady := FALSE;
	tObjectID := 16#FFFFFFFF;

ELSE
	(* clear error flag *)
	nErrorId := BACnet_ERR_NO_ERROR;
	(* ready state *)
	bReady := TRUE;
	(* present value *)
	bPresentValue := _PresentValue;
	tObjectID := _ObjectId;

END_IF

(* set error flag *)
bError := (nErrorId <> BACnet_ERR_NO_ERROR);
END_FUNCTION_BLOCK

(* POU FB_BACnet_RemoteCalendar_POLL, ST *)
FUNCTION_BLOCK FB_BACnet_RemoteCalendar_POLL
VAR_IN_OUT
	RemoteDevice		: FB_BACnet_RemoteDevice;
END_VAR
VAR_OUTPUT
	bReady				: BOOL;
	bPresentValue		: BOOL;
	bError				: BOOL;
	nErrorId			: UINT;
END_VAR
VAR
	_PresentValue AT%I*: BOOL;	(* ~(BACnet_PresentValue 				:		: )
									(BACnet_ObjectType 					: CAL	: )
									(BACnet_RemoteCycletimeRead 		: 5000	: )
									(BACnet_RemoteFlagsRead        		: 2		: )
                            		(BACnet_RemoteCycleTimeWrite   		: 1000	: )
                            		(BACnet_RemoteFlagsWrite       		: 1		: )	*)
	_nUpdateCount : UDINT := 0;
END_VAR
(* update client device *)
IF RemoteDevice._nUpdateCount = _nUpdateCount THEN
	RemoteDevice();
END_IF
(* remind current number of update counter *)
_nUpdateCount := RemoteDevice._nUpdateCount;

IF RemoteDevice.bOperational THEN
	(* clear error flag *)
	nErrorId := BACnet_ERR_NO_ERROR;
	(* ready state *)
	bReady := TRUE;
	(* present value *)
	bPresentValue := _PresentValue;
ELSE
	(* server device not ready, reset local ready also *)
	bReady := FALSE;
	(* and set error ID *)
	nErrorId := BACnet_ERR_OPERATIONAL;
END_IF

(* set error flag *)
bError := (nErrorId <> BACnet_ERR_NO_ERROR);
END_FUNCTION_BLOCK

(* POU FB_BACnet_RemoteCommand, ST *)
FUNCTION_BLOCK FB_BACnet_RemoteCommand
VAR_INPUT
	bEnablePV			: BOOL;
	nPV					: UDINT;
	bRetrigger			: BOOL; (* execute selected action on raising edge again *)
END_VAR
VAR_IN_OUT
	RemoteDevice		: FB_BACnet_RemoteDevice;
END_VAR
VAR_OUTPUT
	bReady				: BOOL;
	nPresentValue		: UDINT;
	bAllWritesOk		: BOOL; (* all actions in selected action list are written *)
	bInProcess			: BOOL; (* object is busy *)
	bError				: BOOL;
	nErrorId			: UINT;
END_VAR
VAR
	_PresentValueIn AT%I*: UDINT; 		(* ~(BACnet_PresentValue 				:		: )
								   			(BACnet_ObjectType 					: CMD	: )
											(BACnet_RemoteCycletimeRead 		: 1000	: )
											(BACnet_RemoteFlagsRead        		: 1		: )
											(BACnet_RemoteResubscriptionInterval: 240	: )
	                                		(BACnet_RemoteCycleTimeWrite   		: 1000	: )
	                                		(BACnet_RemoteFlagsWrite       		: 1		: )	*)
	_InProcess AT%I*: BOOL;				(* ~(BACnet_InProcess 					:		: )	*)
	_AllWritesSuccessful AT%I*: BOOL;	(* ~(BACnet_AllWritesSuccessful			:		: )	*)
    _PresentValueOut AT%Q*: UDINT;		(* ~(BACnet_PresentValue	 	   		:      	: )	*)
	_nUpdateCount : UDINT := 0;
	_rtrigRetriggerPv : R_TRIG;
END_VAR
(* update client device *)
IF RemoteDevice._nUpdateCount = _nUpdateCount THEN
	RemoteDevice();
END_IF
(* remind current number of update counter *)
_nUpdateCount := RemoteDevice._nUpdateCount;

(* call trigger *)
_rtrigRetriggerPv(CLK:= bRetrigger, Q=> );

IF RemoteDevice.bOperational THEN
	(* clear error flag *)
	nErrorId := BACnet_ERR_NO_ERROR;
	(* ready state *)
	bReady := TRUE;
	(* present value from BACnet *)
	nPresentValue := _PresentValueIn;
	(* present value to BACnet *)
	IF bEnablePV THEN
		IF _rtrigRetriggerPv.Q THEN
			(* trigger action list *)
			_PresentValueOut := 0;
		ELSE
			(* set present value *)
			_PresentValueOut := nPV;
		END_IF
	ELSE
		(* deactivate mapped present value --> other objects can write to property *)
		_PresentValueOut := 16#FFFFFFFF;
	END_IF
	(* other states *)
	bAllWritesOk := _AllWritesSuccessful;
	bInProcess := _InProcess;
ELSIF RemoteDevice.bFirstCycle THEN
	(* first call of the server device since reboot/reset *)
	bReady := FALSE;
	_PresentValueOut := 0;
ELSE
	(* server device not ready, reset local ready also *)
	bReady := FALSE;
	(* and set error ID *)
	nErrorId := BACnet_ERR_WRONG_MAPPING;
END_IF

(* set error flag *)
bError := (nErrorId <> BACnet_ERR_NO_ERROR);
END_FUNCTION_BLOCK

(* POU FB_BACnet_RemoteCommand_EX, ST *)
FUNCTION_BLOCK FB_BACnet_RemoteCommand_EX
VAR_INPUT
	bEnablePV			: BOOL;
	nPV					: UDINT;
	bRetrigger			: BOOL; (* execute selected action on raising edge again *)
END_VAR
VAR_IN_OUT
	RemoteDevice		: FB_BACnet_RemoteDevice;
END_VAR
VAR_OUTPUT
	bReady				: BOOL;
	nPresentValue		: UDINT;
	bAllWritesOk		: BOOL; (* all actions in selected action list are written *)
	bInProcess			: BOOL; (* object is busy *)
	tObjectID			: T_BACnet_ObjectIdentifier := 16#FFFFFFFF;
	bError				: BOOL;
	nErrorId			: UINT;
END_VAR
VAR
	_PresentValueIn AT%I*: UDINT; 		(* ~(BACnet_PresentValue 				:		: )
								   			(BACnet_ObjectType 					: CMD	: )
											(BACnet_RemoteCycletimeRead 		: 1000	: )
											(BACnet_RemoteFlagsRead        		: 1		: )
											(BACnet_RemoteResubscriptionInterval: 240	: )
	                                		(BACnet_RemoteCycleTimeWrite   		: 1000	: )
	                                		(BACnet_RemoteFlagsWrite       		: 1		: )	*)
	_ObjectId AT%I*: DWORD;				(* ~(BACnet_ObjectIdentifier			:		: LINK) *)
	_InProcess AT%I*: BOOL;				(* ~(BACnet_InProcess 					:		: )	*)
	_AllWritesSuccessful AT%I*: BOOL;	(* ~(BACnet_AllWritesSuccessful			:		: )	*)
    _PresentValueOut AT%Q*: UDINT;		(* ~(BACnet_PresentValue	 	   		:      	: )	*)
	_nUpdateCount : UDINT := 0;
	_rtrigRetriggerPv : R_TRIG;
	_bRetriggerReq : BOOL;
END_VAR
(* update client device *)
IF RemoteDevice._nUpdateCount = _nUpdateCount THEN
	RemoteDevice();
END_IF
(* remind current number of update counter *)
_nUpdateCount := RemoteDevice._nUpdateCount;

(* call trigger *)
_rtrigRetriggerPv(CLK:= bRetrigger, Q=> );

IF RemoteDevice.bFirstCycle THEN
	(* first call of the server device since reboot/reset *)
	bReady := FALSE;
	_PresentValueOut := 0;
	_bRetriggerReq := FALSE;

ELSIF NOT RemoteDevice.bOperational THEN
	(* server device not ready, reset local ready also *)
	bReady := FALSE;
	(* and set error ID *)
	nErrorId := BACnet_ERR_WRONG_MAPPING;
	_bRetriggerReq := FALSE;

ELSIF (F_BACnet_GetObjType(_ObjectId) <> BACnetObjectType_Command) THEN
	(* wrong mapping / invalid object ID *)
	IF _ObjectId = 0 THEN
		nErrorId := BACnet_ERR_WRONG_MAPPING;
	ELSE
		nErrorId := BACnet_ERR_INVALID_OBJECTID;
	END_IF
	bReady := FALSE;
	tObjectID := 16#FFFFFFFF;
	_bRetriggerReq := FALSE;

ELSE
	(* object ID *)
	tObjectID := _ObjectId;
	(* clear error flag *)
	nErrorId := BACnet_ERR_NO_ERROR;
	(* activities *)
	bAllWritesOk := _AllWritesSuccessful;
	bInProcess := _InProcess;
	(* ready state *)
	bReady := TRUE;
	(* present value from BACnet *)
	nPresentValue := _PresentValueIn;
	(* present value to BACnet *)
	IF bEnablePV THEN
		IF (NOT bInProcess) THEN
			IF _bRetriggerReq THEN
				(* trigger action list *)
				_PresentValueOut := 0;
			ELSE
				(* set present value *)
				_PresentValueOut := nPV;
			END_IF
			_bRetriggerReq := FALSE;
		END_IF
	ELSE
		(* deactivate mapped present value --> other objects can write to property *)
		_PresentValueOut := 16#FFFFFFFF;
		_bRetriggerReq := FALSE;
	END_IF

END_IF

(* set error flag *)
bError := (nErrorId <> BACnet_ERR_NO_ERROR);
END_FUNCTION_BLOCK

(* POU FB_BACnet_RemoteCommand_POLL, ST *)
FUNCTION_BLOCK FB_BACnet_RemoteCommand_POLL
VAR_INPUT
	bEnablePV			: BOOL;
	nPV					: UDINT;
	bRetrigger			: BOOL; (* execute selected action on raising edge again *)
END_VAR
VAR_IN_OUT
	RemoteDevice		: FB_BACnet_RemoteDevice;
END_VAR
VAR_OUTPUT
	bReady				: BOOL;
	nPresentValue		: UDINT;
	bAllWritesOk		: BOOL; (* all actions in selected action list are written *)
	bInProcess			: BOOL; (* object is busy *)
	bError				: BOOL;
	nErrorId			: UINT;
END_VAR
VAR
	_PresentValueIn AT%I*: UDINT; 		(* ~(BACnet_PresentValue 				:		: )
								   			(BACnet_ObjectType 					: CMD	: )
											(BACnet_RemoteCycletimeRead 		: 5000	: )
											(BACnet_RemoteFlagsRead        		: 2		: )
	                                		(BACnet_RemoteCycleTimeWrite   		: 1000	: )
	                                		(BACnet_RemoteFlagsWrite       		: 1		: )	*)
	_InProcess AT%I*: BOOL;				(* ~(BACnet_InProcess 					:		: )	*)
	_AllWritesSuccessful AT%I*: BOOL;	(* ~(BACnet_AllWritesSuccessful			:		: )	*)
    _PresentValueOut AT%Q*: UDINT;		(* ~(BACnet_PresentValue	 	   		:      	: )	*)
	_nUpdateCount : UDINT := 0;
	_rtrigRetriggerPv : R_TRIG;
END_VAR
(* update client device *)
IF RemoteDevice._nUpdateCount = _nUpdateCount THEN
	RemoteDevice();
END_IF
(* remind current number of update counter *)
_nUpdateCount := RemoteDevice._nUpdateCount;

(* call trigger *)
_rtrigRetriggerPv(CLK:= bRetrigger, Q=> );

IF RemoteDevice.bOperational THEN
	(* clear error flag *)
	nErrorId := BACnet_ERR_NO_ERROR;
	(* ready state *)
	bReady := TRUE;
	(* present value from BACnet *)
	nPresentValue := _PresentValueIn;
	(* present value to BACnet *)
	IF bEnablePV THEN
		IF _rtrigRetriggerPv.Q THEN
			(* trigger action list *)
			_PresentValueOut := 0;
		ELSE
			(* set present value *)
			_PresentValueOut := nPV;
		END_IF
	ELSE
		(* deactivate mapped present value --> other objects can write to property *)
		_PresentValueOut := 16#FFFFFFFF;
	END_IF
	(* other states *)
	bAllWritesOk := _AllWritesSuccessful;
	bInProcess := _InProcess;
ELSIF RemoteDevice.bFirstCycle THEN
	(* first call of the server device since reboot/reset *)
	bReady := FALSE;
	_PresentValueOut := 0;
ELSE
	(* server device not ready, reset local ready also *)
	bReady := FALSE;
	(* and set error ID *)
	nErrorId := BACnet_ERR_WRONG_MAPPING;
END_IF

(* set error flag *)
bError := (nErrorId <> BACnet_ERR_NO_ERROR);
END_FUNCTION_BLOCK

(* POU FB_BACnet_RemoteDevice_POLL, ST *)
FUNCTION_BLOCK FB_BACnet_RemoteDevice_POLL
VAR_INPUT
	bReset				: BOOL;
	bAutoReset			: BOOL;
	bDisableWOC			: BOOL;
	bReSubscribeCOV		: BOOL;
	bAutoReSubscribe	: BOOL;
	bTriggerWOC			: BOOL; (* Revision 9 feature: FALSE --> TRUE writes all output process data to remote device *)
	nAmsPort			: UINT := 0; (* Optional setting: AMS port of BACnet client, default = not set *)
END_VAR
VAR_OUTPUT
	stAdsConn			: ST_BACnet_AdsConnection;
	eSystemStatus		: E_BACNETDEVICESTATUS;
	bEthLinkOk			: BOOL;
	bGatewayOk			: BOOL;
	sAmsNetId			: T_AmsNetId;
	bEnabledWOC			: BOOL;
	bWOCTriggered		: BOOL;
	bOperational		: BOOL;
	bConnecting			: BOOL;
	bFirstCycle			: BOOL;
	bError				: BOOL;
	nErrorId			: UINT;
	bClientTimeout		: BOOL;
	bServiceFailed		: BOOL;
	nTimeoutCnt			: UDINT;
	nServiceFailCnt		: UDINT;
END_VAR
VAR
	_ObjectId AT%I*:DWORD;			(* ~(BACnet_ObjectIdentifier			:		: LINK ) *)
	_SystemStatus AT%I*	: E_BACNETDEVICESTATUS;	(* ~
										(BACnet_SystemStatus 				: 		: )
										(BACnet_ObjectType					: DEV	: )
										(BACnet_RemoteCycletimeRead 		: 5000	: )
										(BACnet_RemoteFlagsRead        		: 2     : )
										(BACnet_RemoteCycleTimeWrite   		: 1000	: )
										(BACnet_RemoteFlagsWrite       		: 1		: ) *)
	_ClientStatus AT%I*:WORD;		(* ~(BACnet_ClientStatus				:		: )	*)
	_ClientControl AT%Q*:WORD;		(* ~(BACnet_ClientControl				:		: ) *)
	_rtrigReset			: R_TRIG;
	_rtrigOperational	: R_TRIG;
	_rtrigResubscribe	: R_TRIG;
	_rtrigTimeoutCnt	: R_TRIG;
	_rtrigServiceFailCnt: R_TRIG;
	_bReqResubscribe	: BOOL;
	_bComplete			: BOOL;
	_tofTimeoutLeft		: TOF;
	_tofServiceErrLeft	: TOF;
	_ftrigTimeoutLeft	: F_TRIG;

	_bHasStarted		: BOOL := TRUE;
	_nUpdateCount		: UDINT := 0;
	_nUpdateCountAdp 	: UDINT := 0;
	_BACnetAdapter		: POINTER TO FB_BACnet_Adapter;
	_AdsConn			: _FB_BACnet_AdsConn;
	_bLegacyMode		: BOOL;
	_tonAdsReset		: TON;

	_rtrigWOC			: R_TRIG;
	_bTriggerWOC		: BOOL;
	_tonWOCTrigger		: TON;
END_VAR
(* check pointer to bacnet adapter instance *)
IF pBACnet_Adapter > 0 THEN
	_BACnetAdapter := pBACnet_Adapter;
ELSE
	_BACnetAdapter := ADR(fbBACnet_Adapter);
END_IF

(* update server device *)
IF _BACnetAdapter^._nUpdateCount = _nUpdateCountAdp THEN
	_BACnetAdapter^();
END_IF
(* remind current number of update counter *)
_nUpdateCountAdp := _BACnetAdapter^._nUpdateCount;

(* check for client errors *)
_rtrigTimeoutCnt(CLK:= _ClientStatus.0, Q=> );
IF _rtrigTimeoutCnt.Q AND _bComplete THEN
	nErrorId := BACnet_ERR_CLIENT_TIMEOUT;
ELSIF (NOT _ClientStatus.0) THEN
	(* reset acknowledge flag *)
	_ClientControl.0 := FALSE;
END_IF
_rtrigServiceFailCnt(CLK:= _ClientStatus.1, Q=> );
IF _rtrigServiceFailCnt.Q AND _bComplete THEN
	nErrorId := BACnet_ERR_CLIENT_SERVICE;
ELSIF (NOT _ClientStatus.1) THEN
	(* reset acknowledge flag *)
	_ClientControl.1 := FALSE;
END_IF

(* convert SystemStatus to enumeration *)
eSystemStatus := _SystemStatus;
(* reset trigger *)
_rtrigReset(CLK:= bReset, Q=> );
(* reset error ID and flag *)
IF (nErrorId < 20) OR _rtrigReset.Q OR bAutoReset THEN
	nErrorId := BACnet_ERR_NO_ERROR;
END_IF
IF _rtrigReset.Q OR (NOT _bComplete) OR bAutoReset THEN
	_ClientControl.0 := _ClientStatus.0;
	_ClientControl.1 := _ClientStatus.1;
END_IF

(* read NetId and convert to string *)
sAmsNetId := _BACnetAdapter^.sAmsNetId;
(* check if it plausible *)
IF sAmsNetId = '' THEN
	(* NetId not OK, return with error *)
	nErrorId := BACnet_ERR_NO_VALID_NET_ID;
ELSIF (NOT _BACnetAdapter^.bEthLinkOk) THEN
	(* ethernet link missing *)
	nErrorId := BACnet_ERR_NO_ETH_LINK;
ELSIF (NOT _BACnetAdapter^.bGatewayOk) THEN
	(* gateway missing *)
	nErrorId := BACnet_ERR_NO_GATEWAY;
END_IF

(* summerize timeout errors *)
_tofTimeoutLeft(
	IN:= (_rtrigTimeoutCnt.Q AND _bComplete),
	PT:= T#20s,
	Q=> bClientTimeout,
	ET=> );
IF _tofTimeoutLeft.IN THEN
	nTimeoutCnt := nTimeoutCnt + 1;
END_IF
_ftrigTimeoutLeft(CLK:= _tofTimeoutLeft.Q, Q=> );

(* summerize service errors *)
_tofServiceErrLeft(
	IN:= (_rtrigServiceFailCnt.Q AND _bComplete),
	PT:= T#20s,
	Q=> bServiceFailed,
	ET=> );
IF _tofServiceErrLeft.IN THEN
	nServiceFailCnt := nServiceFailCnt + 1;
END_IF

(* WOC trigger control *)
_rtrigWOC(CLK:= bTriggerWOC, Q=> );
IF (_ClientStatus.2 OR bDisableWOC) AND bTriggerWOC THEN
	nErrorId := BACnet_ERR_WOC_DISABLED;
	_bTriggerWOC := FALSE;
ELSIF _ClientStatus.4 OR _bTriggerWOC THEN
	IF _rtrigWOC.Q THEN
		nErrorId := BACnet_ERR_WOC_TRIGGER_ACTIVE;
	ELSIF (NOT bTriggerWOC) THEN
		_bTriggerWOC := FALSE;
	END_IF
ELSIF _rtrigWOC.Q THEN
	_bTriggerWOC := TRUE;
END_IF

(* controls *)
_ClientControl.2 := bDisableWOC;
_ClientControl.3 := _bReqResubscribe;
_ClientControl.4 := _bTriggerWOC;

(* states *)
bEthLinkOk := _BACnetAdapter^.bEthLinkOk;
bGatewayOk := _BACnetAdapter^.bGatewayOk;

bEnabledWOC := (NOT _ClientStatus.2);
bConnecting := (SHR((_ClientStatus AND 16#FF00), 8) < 4);
_bComplete :=		(NOT bConnecting)
				AND	(_SystemStatus = 0)
				AND	_BACnetAdapter^.bEthLinkOk;
bOperational :=		_bComplete
				AND ((NOT _ClientStatus.0) OR bAutoReset);
bWOCTriggered	:= bTriggerWOC AND _ClientStatus.4 AND (NOT (_ClientStatus.2 OR bDisableWOC));

(* Resubscribe COV *)
_rtrigOperational(CLK:= bOperational, Q=> );
_rtrigResubscribe(CLK:= bReSubscribeCOV, Q=> );
IF		(		(		(		_rtrigOperational.Q
							OR (_ftrigTimeoutLeft.Q AND bAutoReset)
						)
					AND	bAutoReSubscribe
				)
			OR	_rtrigResubscribe.Q
		)
	AND	(NOT _bReqResubscribe)
THEN
	(* operation mode reached or resubscription was externally triggered, start resubcription *)
	_bReqResubscribe	:= TRUE;
ELSIF (NOT bOperational) THEN
	(* not operational *)
	_bReqResubscribe	:= FALSE;
ELSE
	IF _bReqResubscribe AND _ClientStatus.3 THEN
		(* resubscription triggered *)
		_bReqResubscribe := FALSE;
	END_IF
END_IF

